KUKA KRL program: MyProgram_076().src

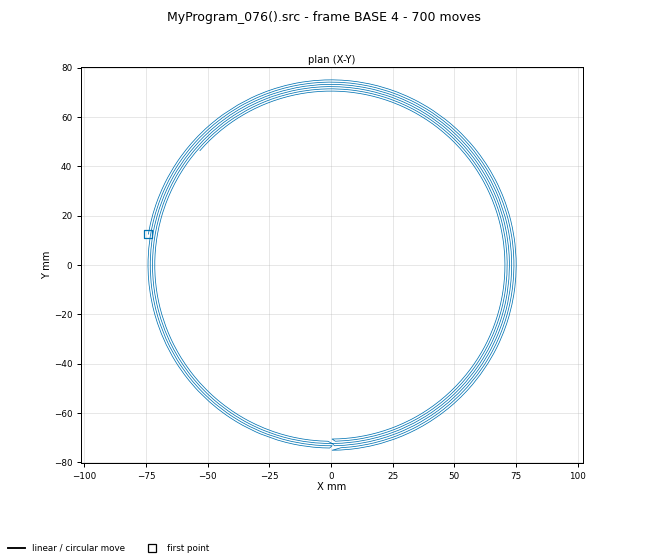
[picture p0: tool path of MyProgram_076().src in frame BASE 4, 700 of 700 moves have a stored position in this frame; points joined in program order, loops and branches not executed]
&ACCESS RVP
&REL 1
&PARAM TEMPLATE = C:\KRC\Roboter\Template\vorgabe
&PARAM EDITMASK = *
DEF MyProgram_076()
; ---- Setting reference (Base) ----
$BASE = BASE_DATA[4]

; --------------------------
; ---- Setting tool (TCP) ----
$TOOL = TOOL_DATA[3]
; --------------------------

$VEL.CP = VEL_APROX_PRINT
Startdeposition()
$VEL.CP = VEL_PRINT
LIN {X -74.0338,Y 12.5414,Z 79,A 163.3796,B 24.8998,C -2.3111,E1 24.8428,E2 281.1922} C_DIS
LIN {X -73.2521,Y 16.5095,Z 79,A 161.2903,B 24.8969,C -2.3435,E1 24.844,E2 283.2162} C_DIS
LIN {X -72.1494,Y 20.8052,Z 79,A 158.1049,B 24.8956,C -2.3587,E1 24.8463,E2 286.3839} C_DIS
LIN {X -70.9389,Y 24.6173,Z 79,A 155.0379,B 24.8948,C -2.3677,E1 24.8489,E2 289.4469} C_DIS
LIN {X -70.0447,Y 27.057,Z 79,A 152.3998,B 24.8956,C -2.3586,E1 24.8515,E2 292.1217} C_DIS
LIN {X -68.6085,Y 30.5169,Z 79,A 149.1898,B 24.8956,C -2.3591,E1 24.8551,E2 295.3482} C_DIS
LIN {X -67.2388,Y 33.425,Z 79,A 147.2866,B 24.8938,C -2.379,E1 24.8574,E2 297.2143} C_DIS
LIN {X -66.1724,Y 35.491,Z 79,A 145.1905,B 24.894,C -2.3766,E1 24.8602,E2 299.3271} C_DIS
LIN {X -63.8148,Y 39.5728,Z 79,A 141.9536,B 24.8923,C -2.3952,E1 24.8648,E2 302.5364} C_DIS
LIN {X -62.0519,Y 42.2834,Z 79,A 139.6485,B 24.8914,C -2.4058,E1 24.8683,E2 304.8278} C_DIS
LIN {X -60.8028,Y 44.0616,Z 79,A 137.7393,B 24.8915,C -2.4043,E1 24.8714,E2 306.7497} C_DIS
LIN {X -58.7303,Y 46.7866,Z 79,A 135.0507,B 24.8911,C -2.4094,E1 24.876,E2 309.4388} C_DIS
LIN {X -56.5657,Y 49.3821,Z 79,A 132.3745,B 24.8907,C -2.4137,E1 24.8809,E2 312.1171} C_DIS
LIN {X -53.9325,Y 52.2455,Z 79,A 129.4614,B 24.8899,C -2.4222,E1 24.8864,E2 315.0225} C_DIS
LIN {X -50.9748,Y 55.1346,Z 79,A 126.5258,B 24.8887,C -2.4348,E1 24.8923,E2 317.9402} C_DIS
LIN {X -49.0445,Y 56.8585,Z 79,A 124.2457,B 24.889,C -2.432,E1 24.8972,E2 320.2362} C_DIS
LIN {X -45.9844,Y 59.3611,Z 79,A 121.4566,B 24.8879,C -2.4439,E1 24.9032,E2 323.0073} C_DIS
LIN {X -43.6877,Y 61.071,Z 79,A 118.8455,B 24.8884,C -2.438,E1 24.9092,E2 325.6414} C_DIS
LIN {X -37.719,Y 64.9268,Z 79,A 113.8884,B 24.8865,C -2.4594,E1 24.9208,E2 330.5633} C_DIS
LIN {X -32.3398,Y 67.7676,Z 79,A 109.0548,B 24.8862,C -2.4622,E1 24.9328,E2 335.4033} C_DIS
LIN {X -30.0073,Y 68.8319,Z 79,A 106.5716,B 24.8871,C -2.4521,E1 24.9392,E2 337.9164} C_DIS
LIN {X -26.1038,Y 70.4061,Z 79,A 103.4974,B 24.8864,C -2.4597,E1 24.9472,E2 340.979} C_DIS
LIN {X -22.65,Y 71.5922,Z 79,A 100.0527,B 24.8877,C -2.4467,E1 24.9565,E2 344.461} C_DIS
LIN {X -18.3648,Y 72.8088,Z 79,A 96.6299,B 24.8874,C -2.4494,E1 24.9657,E2 347.8821} C_DIS
LIN {X -13.9688,Y 73.778,Z 79,A 94.2298,B 24.8847,C -2.4781,E1 24.9721,E2 350.2167} C_DIS
LIN {X -11.4549,Y 74.2095,Z 79,A 92.0843,B 24.8851,C -2.4744,E1 24.9781,E2 352.3729} C_DIS
LIN {X -6.9976,Y 74.7617,Z 79,A 87.808,B 24.8869,C -2.4547,E1 24.9901,E2 356.6986} C_DIS
LIN {X -2.4864,Y 75.0475,Z 79,A 85.4114,B 24.8843,C -2.4827,E1 24.9966,E2 359.0291} C_DIS
LIN {X 0.7273,Y 75.0854,Z 79,A 82.8148,B 24.8846,C -2.4794,E1 25.0039,E2 361.6334} C_DIS
LIN {X 4.3078,Y 74.9649,Z 79,A 79.597,B 24.8858,C -2.467,E1 25.0129,E2 364.8796} C_DIS
LIN {X 7.625,Y 74.7005,Z 79,A 77.7484,B 24.8841,C -2.4847,E1 25.0179,E2 366.6849} C_DIS
LIN {X 11.0283,Y 74.2755,Z 79,A 74.5426,B 24.8856,C -2.4686,E1 25.0269,E2 369.9263} C_DIS
LIN {X 15.5826,Y 73.4542,Z 79,A 71.3552,B 24.8849,C -2.4762,E1 25.0356,E2 373.0918} C_DIS
LIN {X 19.0638,Y 72.6291,Z 79,A 68.6928,B 24.8849,C -2.4764,E1 25.0428,E2 375.7498} C_DIS
LIN {X 23.5565,Y 71.2992,Z 79,A 65.0604,B 24.8853,C -2.4722,E1 25.0525,E2 379.3857} C_DIS
LIN {X 26.7438,Y 70.1646,Z 79,A 61.6181,B 24.8877,C -2.4466,E1 25.0616,E2 382.8812} C_DIS
LIN {X 30.9008,Y 68.4355,Z 79,A 59.2126,B 24.8854,C -2.4707,E1 25.0676,E2 385.2236} C_DIS
LIN {X 33.9507,Y 66.9752,Z 79,A 56.6895,B 24.8856,C -2.4691,E1 25.0739,E2 387.7438} C_DIS
LIN {X 35.7546,Y 66.0294,Z 79,A 54.9592,B 24.8862,C -2.4622,E1 25.0782,E2 389.4855} C_DIS
LIN {X 39.1193,Y 64.0934,Z 79,A 52.1395,B 24.8862,C -2.4619,E1 25.0849,E2 392.2974} C_DIS
LIN {X 41.3094,Y 62.7041,Z 79,A 49.8554,B 24.8873,C -2.4503,E1 25.0903,E2 394.6014} C_DIS
LIN {X 46.3215,Y 59.0989,Z 79,A 45.5003,B 24.8872,C -2.4521,E1 25.1001,E2 398.9366} C_DIS
LIN {X 48.4243,Y 57.3889,Z 79,A 42.7997,B 24.8891,C -2.4304,E1 25.1059,E2 401.6781} C_DIS
LIN {X 50.9296,Y 55.1769,Z 79,A 40.8978,B 24.8879,C -2.4436,E1 25.1098,E2 403.5411} C_DIS
LIN {X 52.8577,Y 53.3324,Z 79,A 38.5166,B 24.8892,C -2.4296,E1 25.1145,E2 405.9455} C_DIS
LIN {X 56.4292,Y 49.5384,Z 79,A 34.9262,B 24.889,C -2.4318,E1 25.1213,E2 409.5149} C_DIS
LIN {X 58.3316,Y 47.2832,Z 79,A 32.0216,B 24.8912,C -2.4079,E1 25.1265,E2 412.4626} C_DIS
LIN {X 60.4304,Y 44.5702,Z 79,A 29.7878,B 24.8908,C -2.4125,E1 25.1302,E2 414.6748} C_DIS
LIN {X 62.9223,Y 40.9777,Z 79,A 26.7139,B 24.8908,C -2.4116,E1 25.1349,E2 417.7354} C_DIS
LIN {X 64.6181,Y 38.2462,Z 79,A 23.7768,B 24.8927,C -2.3912,E1 25.1392,E2 420.7057} C_DIS
LIN {X 66.7813,Y 34.3302,Z 79,A 20.9154,B 24.8921,C -2.398,E1 25.1429,E2 423.536} C_DIS
LIN {X 67.7546,Y 32.3668,Z 79,A 19.0536,B 24.893,C -2.3878,E1 25.1452,E2 425.4119} C_DIS
LIN {X 69.485,Y 28.4629,Z 79,A 15.3261,B 24.8951,C -2.3649,E1 25.1493,E2 429.1731} C_DIS
LIN {X 70.7518,Y 25.1506,Z 79,A 13.3493,B 24.8939,C -2.3783,E1 25.1511,E2 431.1071} C_DIS
LIN {X 72.1899,Y 20.6623,Z 79,A 9.7524,B 24.8948,C -2.3676,E1 25.1541,E2 434.7089} C_DIS
LIN {X 72.8382,Y 18.2504,Z 79,A 7.2574,B 24.8969,C -2.3445,E1 25.1558,E2 437.2441} C_DIS
LIN {X 73.5531,Y 15.1069,Z 79,A 4.9587,B 24.8971,C -2.3417,E1 25.1571,E2 439.536} C_DIS
LIN {X 74.3323,Y 10.6297,Z 79,A 1.971,B 24.8968,C -2.3451,E1 25.1584,E2 442.4982} C_DIS
LIN {X 74.5961,Y 8.5861,Z 79,A 0.0072,B 24.8983,C -2.3286,E1 25.159,E2 444.4893} C_DIS
LIN {X 75.0392,Y 2.7571,Z 79,A -4.02,B 24.8983,C -2.3273,E1 25.1597,E2 448.4957} C_DIS
LIN {X 75.0885,Y -0.2198,Z 79,A -6.074,B 24.8984,C -2.3266,E1 25.1597,E2 450.5391} C_DIS
LIN {X 74.9286,Y -4.8989,Z 79,A -10.2294,B 24.9009,C -2.2979,E1 25.1592,E2 454.7376} C_DIS
LIN {X 74.5301,Y -9.1497,Z 79,A -13.0627,B 24.9007,C -2.3001,E1 25.1584,E2 457.549} C_DIS
LIN {X 74.0928,Y -12.1884,Z 79,A -15.2797,B 24.9011,C -2.2964,E1 25.1575,E2 459.7616} C_DIS
LIN {X 73.3464,Y -16.0806,Z 79,A -18.5241,B 24.9024,C -2.2803,E1 25.1556,E2 463.0251} C_DIS
LIN {X 72.2095,Y -20.593,Z 79,A -21.5023,B 24.9019,C -2.2862,E1 25.1536,E2 465.9721} C_DIS
LIN {X 71.233,Y -23.7528,Z 79,A -24.7017,B 24.9043,C -2.2583,E1 25.1508,E2 469.2193} C_DIS
LIN {X 69.9926,Y -27.1916,Z 79,A -27.419,B 24.9049,C -2.2519,E1 25.1481,E2 471.9366} C_DIS
LIN {X 68.3546,Y -31.0804,Z 79,A -30.3314,B 24.9049,C -2.2513,E1 25.1449,E2 474.8343} C_DIS
LIN {X 67.0986,Y -33.7059,Z 79,A -32.5046,B 24.9054,C -2.2462,E1 25.1422,E2 477.0081} C_DIS
LIN {X 65.901,Y -35.9913,Z 79,A -34.7495,B 24.9065,C -2.2323,E1 25.1392,E2 479.274} C_DIS
LIN {X 63.5951,Y -39.9245,Z 79,A -37.8445,B 24.9064,C -2.2337,E1 25.1348,E2 482.3497} C_DIS
LIN {X 60.5065,Y -44.4663,Z 79,A -42.0028,B 24.9073,C -2.2232,E1 25.1282,E2 486.5126} C_DIS
LIN {X 57.3809,Y -48.4337,Z 79,A -46.0102,B 24.9085,C -2.2086,E1 25.1212,E2 490.5358} C_DIS
LIN {X 55.3733,Y -50.7157,Z 79,A -48.5588,B 24.9095,C -2.1961,E1 25.1164,E2 493.1027} C_DIS
LIN {X 52.6657,Y -53.5221,Z 79,A -51.2668,B 24.9095,C -2.1966,E1 25.1111,E2 495.7979} C_DIS
LIN {X 49.7882,Y -56.21,Z 79,A -54.281,B 24.9101,C -2.1894,E1 25.1049,E2 498.817} C_DIS
LIN {X 47.4391,Y -58.2052,Z 79,A -56.8567,B 24.911,C -2.1778,E1 25.0993,E2 501.4103} C_DIS
LIN {X 44.4713,Y -60.5028,Z 79,A -59.6425,B 24.9113,C -2.174,E1 25.0931,E2 504.1949} C_DIS
LIN {X 40.3486,Y -63.3271,Z 79,A -63.2381,B 24.9114,C -2.1728,E1 25.0847,E2 507.7815} C_DIS
LIN {X 37.2123,Y -65.2193,Z 79,A -66.1227,B 24.9121,C -2.1652,E1 25.0778,E2 510.6753} C_DIS
LIN {X 34.3967,Y -66.7473,Z 79,A -68.4125,B 24.9121,C -2.1654,E1 25.0721,E2 512.9579} C_DIS
LIN {X 31.8505,Y -67.9989,Z 79,A -70.53,B 24.9122,C -2.1633,E1 25.0668,E2 515.0748} C_DIS
LIN {X 28.6942,Y -69.3901,Z 79,A -73.5255,B 24.9134,C -2.1493,E1 25.0591,E2 518.0965} C_DIS
LIN {X 25.511,Y -70.6223,Z 79,A -76.2197,B 24.9138,C -2.1434,E1 25.052,E2 520.7991} C_DIS
LIN {X 20.0691,Y -72.358,Z 79,A -80.4465,B 24.9139,C -2.1421,E1 25.0407,E2 525.0216} C_DIS
LIN {X 15.8281,Y -73.4015,Z 79,A -83.441,B 24.9134,C -2.1482,E1 25.0326,E2 527.9972} C_DIS
LIN {X 11.2138,Y -74.2468,Z 79,A -87.0755,B 24.9138,C -2.144,E1 25.0226,E2 531.638} C_DIS
LIN {X 8.1036,Y -74.6504,Z 79,A -89.4305,B 24.9138,C -2.1435,E1 25.0161,E2 533.9922} C_DIS
LIN {X 3.8663,Y -74.9893,Z 79,A -93.5069,B 24.9157,C -2.1198,E1 25.0045,E2 538.1233} C_DIS
LIN {X 0.4928,Y -75.0785,Z 79,A -93.6611,B 24.9105,C -2.1847,E1 25.0046,E2 538.1233} C_DIS
Enddeposition()
LIN {X 0.4928,Y -75.0785,Z 79,A -93.6611,B 24.9105,C -2.1847,E1 25.0046,E2 538.1233} C_DIS
Startdeposition()
$VEL.CP = VEL_PRINT
LIN {X 4.0815,Y -74.0642,Z 79,A -91.2785,B 24.91,C -2.1904,E1 25.0112,E2 535.7279} C_DIS
LIN {X 8.0955,Y -73.7344,Z 79,A -88.3098,B 24.9102,C -2.1882,E1 25.0195,E2 532.7665} C_DIS
LIN {X 11.0368,Y -73.3515,Z 79,A -85.1411,B 24.908,C -2.2141,E1 25.0284,E2 529.5392} C_DIS
LIN {X 14.9582,Y -72.6527,Z 79,A -83.3262,B 24.9107,C -2.1816,E1 25.0331,E2 527.8034} C_DIS
LIN {X 17.5684,Y -72.066,Z 79,A -80.6303,B 24.9091,C -2.201,E1 25.0406,E2 525.0653} C_DIS
LIN {X 21.3791,Y -71.0295,Z 79,A -77.0856,B 24.9077,C -2.2184,E1 25.0502,E2 521.4856} C_DIS
LIN {X 24.874,Y -69.8824,Z 79,A -75.2446,B 24.9097,C -2.1937,E1 25.0549,E2 519.7068} C_DIS
LIN {X 26.7368,Y -69.1907,Z 79,A -73.4018,B 24.9088,C -2.2044,E1 25.0597,E2 517.8425} C_DIS
LIN {X 30.013,Y -67.8347,Z 79,A -70.6724,B 24.9085,C -2.2081,E1 25.0667,E2 515.1108} C_DIS
LIN {X 33.3671,Y -66.2483,Z 79,A -68.1884,B 24.9091,C -2.2019,E1 25.0729,E2 512.6482} C_DIS
LIN {X 34.9862,Y -65.4087,Z 79,A -66.3095,B 24.9077,C -2.2177,E1 25.0776,E2 510.7373} C_DIS
LIN {X 38.5939,Y -63.3457,Z 79,A -63.4619,B 24.9081,C -2.2131,E1 25.0844,E2 507.9092} C_DIS
LIN {X 40.1525,Y -62.3694,Z 79,A -61.5131,B 24.9066,C -2.231,E1 25.0891,E2 505.9243} C_DIS
LIN {X 43.2174,Y -60.2863,Z 79,A -59.2432,B 24.9076,C -2.2196,E1 25.0942,E2 503.6892} C_DIS
LIN {X 45.6157,Y -58.4925,Z 79,A -56.4487,B 24.906,C -2.2385,E1 25.1005,E2 500.8603} C_DIS
LIN {X 48.7088,Y -55.943,Z 79,A -53.2307,B 24.9051,C -2.2489,E1 25.1073,E2 497.63} C_DIS
LIN {X 52.1516,Y -52.7482,Z 79,A -49.8965,B 24.9051,C -2.2489,E1 25.114,E2 494.3098} C_DIS
LIN {X 55.2474,Y -49.4963,Z 79,A -46.6042,B 24.9048,C -2.2523,E1 25.1203,E2 491.0238} C_DIS
LIN {X 59.3132,Y -44.5433,Z 79,A -41.5957,B 24.9036,C -2.267,E1 25.1291,E2 486.004} C_DIS
LIN {X 61.9752,Y -40.7583,Z 79,A -38.3749,B 24.9036,C -2.2663,E1 25.1341,E2 482.8006} C_DIS
LIN {X 63.2688,Y -38.7198,Z 79,A -35.4397,B 24.9004,C -2.3035,E1 25.1385,E2 479.7924} C_DIS
LIN {X 65.1878,Y -35.3937,Z 79,A -33.2931,B 24.9018,C -2.2875,E1 25.1414,E2 477.6947} C_DIS
LIN {X 66.848,Y -32.1483,Z 79,A -30.413,B 24.9009,C -2.2977,E1 25.1449,E2 474.806} C_DIS
LIN {X 68.2757,Y -28.9936,Z 79,A -27.8103,B 24.9004,C -2.3036,E1 25.1478,E2 472.2036} C_DIS
LIN {X 69.318,Y -26.4046,Z 79,A -25.8859,B 24.9004,C -2.3033,E1 25.1498,E2 470.2906} C_DIS
LIN {X 70.6962,Y -22.4547,Z 79,A -22.6503,B 24.8996,C -2.3133,E1 25.1527,E2 467.0496} C_DIS
LIN {X 71.4938,Y -19.7737,Z 79,A -20.1823,B 24.8982,C -2.3293,E1 25.1546,E2 464.558} C_DIS
LIN {X 72.4055,Y -16.1152,Z 79,A -16.8313,B 24.8962,C -2.3517,E1 25.1567,E2 461.1737} C_DIS
LIN {X 73.0556,Y -12.8498,Z 79,A -15.2572,B 24.8982,C -2.3298,E1 25.1575,E2 459.6603} C_DIS
LIN {X 73.5866,Y -9.3387,Z 79,A -11.8884,B 24.8957,C -2.3573,E1 25.1588,E2 456.2465} C_DIS
LIN {X 74.0023,Y -5.0821,Z 79,A -7.8424,B 24.8928,C -2.3903,E1 25.1597,E2 452.1466} C_DIS
LIN {X 74.1745,Y -0.5549,Z 79,A -5.6994,B 24.8954,C -2.3605,E1 25.1597,E2 450.0866} C_DIS
LIN {X 74.1537,Y 1.884,Z 79,A -2.7613,B 24.8921,C -2.3982,E1 25.1596,E2 447.0771} C_DIS
LIN {X 73.9615,Y 5.6506,Z 79,A -0.6692,B 24.8935,C -2.3826,E1 25.1592,E2 445.034} C_DIS
LIN {X 73.6238,Y 9.0483,Z 79,A 1.7052,B 24.8935,C -2.383,E1 25.1585,E2 442.6727} C_DIS
LIN {X 73.2988,Y 11.3776,Z 79,A 3.9459,B 24.8918,C -2.4014,E1 25.1575,E2 440.4019} C_DIS
LIN {X 72.654,Y 14.9521,Z 79,A 6.6534,B 24.8913,C -2.4071,E1 25.1561,E2 437.6968} C_DIS
LIN {X 71.7299,Y 18.8993,Z 79,A 9.4116,B 24.8914,C -2.4055,E1 25.1543,E2 434.9583} C_DIS
LIN {X 70.995,Y 21.4902,Z 79,A 12.4708,B 24.8882,C -2.4409,E1 25.1518,E2 431.8329} C_DIS
LIN {X 69.8305,Y 25.0208,Z 79,A 15.0646,B 24.8882,C -2.4409,E1 25.1493,E2 429.2536} C_DIS
LIN {X 68.3042,Y 28.926,Z 79,A 17.6554,B 24.8891,C -2.431,E1 25.1467,E2 426.7004} C_DIS
LIN {X 66.6033,Y 32.6537,Z 79,A 20.616,B 24.8888,C -2.4339,E1 25.1432,E2 423.7491} C_DIS
LIN {X 65.4425,Y 34.9229,Z 79,A 23.6796,B 24.8854,C -2.4714,E1 25.1391,E2 420.6128} C_DIS
LIN {X 63.5934,Y 38.1864,Z 79,A 25.5376,B 24.8875,C -2.4485,E1 25.1365,E2 418.8186} C_DIS
LIN {X 61.4007,Y 41.6186,Z 79,A 28.8611,B 24.8863,C -2.4617,E1 25.1315,E2 415.4806} C_DIS
LIN {X 57.9026,Y 46.3622,Z 79,A 33.2981,B 24.8856,C -2.4693,E1 25.124,E2 411.0468} C_DIS
LIN {X 56.602,Y 47.9418,Z 79,A 35.7497,B 24.8829,C -2.4982,E1 25.1195,E2 408.538} C_DIS
LIN {X 54.2039,Y 50.6363,Z 79,A 38.0338,B 24.8837,C -2.4897,E1 25.1152,E2 406.2839} C_DIS
LIN {X 51.9222,Y 52.9748,Z 79,A 40.2849,B 24.8839,C -2.4872,E1 25.1108,E2 404.0484} C_DIS
LIN {X 48.6804,Y 55.9679,Z 79,A 44.1161,B 24.8821,C -2.506,E1 25.1027,E2 400.188} C_DIS
LIN {X 45.196,Y 58.8174,Z 79,A 47.4692,B 24.8819,C -2.5087,E1 25.0954,E2 396.8409} C_DIS
LIN {X 41.1343,Y 61.7273,Z 79,A 50.8713,B 24.8825,C -2.5022,E1 25.0877,E2 393.4659} C_DIS
LIN {X 38.8606,Y 63.1836,Z 79,A 53.3129,B 24.8812,C -2.5153,E1 25.0818,E2 391.001} C_DIS
LIN {X 34.5422,Y 65.643,Z 79,A 56.6631,B 24.882,C -2.507,E1 25.0737,E2 387.6805} C_DIS
LIN {X 32.2302,Y 66.8086,Z 79,A 58.7379,B 24.8816,C -2.5115,E1 25.0685,E2 385.6004} C_DIS
LIN {X 27.2296,Y 68.998,Z 79,A 62.9805,B 24.8811,C -2.5166,E1 25.0576,E2 381.3556} C_DIS
LIN {X 23.4337,Y 70.3783,Z 79,A 65.8887,B 24.8814,C -2.5136,E1 25.05,E2 378.4606} C_DIS
LIN {X 18.3849,Y 71.8621,Z 79,A 69.6829,B 24.8818,C -2.5091,E1 25.0399,E2 374.6836} C_DIS
LIN {X 15.2731,Y 72.5867,Z 79,A 72.8346,B 24.88,C -2.5287,E1 25.0312,E2 371.4897} C_DIS
LIN {X 11.7393,Y 73.2412,Z 79,A 75.7304,B 24.8796,C -2.5328,E1 25.0232,E2 368.5871} C_DIS
LIN {X 7.9492,Y 73.7497,Z 79,A 79.408,B 24.8777,C -2.5527,E1 25.0129,E2 364.8648} C_DIS
LIN {X 3.7851,Y 74.0806,Z 79,A 81.4299,B 24.8807,C -2.5207,E1 25.0075,E2 362.9199} C_DIS
LIN {X -0.7943,Y 74.1731,Z 79,A 84.9826,B 24.8807,C -2.5205,E1 24.9976,E2 359.368} C_DIS
LIN {X -4.5442,Y 74.0386,Z 79,A 88.5493,B 24.8792,C -2.5369,E1 24.9875,E2 355.7614} C_DIS
LIN {X -8.3481,Y 73.7058,Z 79,A 91.3267,B 24.8798,C -2.5309,E1 24.9798,E2 352.9967} C_DIS
LIN {X -12.706,Y 73.0815,Z 79,A 94.2335,B 24.8812,C -2.5159,E1 24.9719,E2 350.1231} C_DIS
LIN {X -15.6953,Y 72.4971,Z 79,A 97.1755,B 24.8799,C -2.529,E1 24.9637,E2 347.1464} C_DIS
LIN {X -18.9763,Y 71.7089,Z 79,A 100.1883,B 24.8792,C -2.5368,E1 24.9555,E2 344.1107} C_DIS
LIN {X -22.4216,Y 70.708,Z 79,A 101.9844,B 24.8818,C -2.509,E1 24.9509,E2 342.3777} C_DIS
LIN {X -26.7617,Y 69.1818,Z 79,A 105.6431,B 24.882,C -2.5071,E1 24.9413,E2 338.716} C_DIS
LIN {X -30.2247,Y 67.74,Z 79,A 108.6639,B 24.8821,C -2.506,E1 24.9335,E2 335.6908} C_DIS
LIN {X -35.1702,Y 65.309,Z 79,A 112.9042,B 24.8828,C -2.4988,E1 24.923,E2 331.4564} C_DIS
LIN {X -36.9477,Y 64.3197,Z 79,A 115.711,B 24.8802,C -2.5266,E1 24.916,E2 328.5749} C_DIS
LIN {X -40.9698,Y 61.8358,Z 79,A 117.5481,B 24.885,C -2.4752,E1 24.912,E2 326.8545} C_DIS
LIN {X -43.9498,Y 59.7545,Z 79,A 121.126,B 24.8838,C -2.4882,E1 24.9037,E2 323.2333} C_DIS
LIN {X -47.2986,Y 57.1402,Z 79,A 124.7937,B 24.8836,C -2.4905,E1 24.8957,E2 319.5463} C_DIS
LIN {X -49.7901,Y 54.9844,Z 79,A 127.0934,B 24.8847,C -2.4788,E1 24.891,E2 317.2653} C_DIS
LIN {X -53.273,Y 51.6157,Z 79,A 130.5791,B 24.8861,C -2.4638,E1 24.8841,E2 313.8009} C_DIS
LIN {X -55.111,Y 49.6487,Z 79,A 133.1468,B 24.8855,C -2.4703,E1 24.8792,E2 311.2063} C_DIS
LIN {X -57.2689,Y 47.144,Z 79,A 135.819,B 24.8858,C -2.4665,E1 24.8744,E2 308.5307} C_DIS
LIN {X -60.1199,Y 43.4507,Z 79,A 138.8407,B 24.888,C -2.4431,E1 24.8694,E2 305.5504} C_DIS
LIN {X -62.0554,Y 40.6361,Z 79,A 141.7341,B 24.888,C -2.4419,E1 24.8649,E2 302.6454} C_DIS
LIN {X -64.0387,Y 37.4342,Z 79,A 144.6852,B 24.8888,C -2.4347,E1 24.8607,E2 299.6965} C_DIS
LIN {X -65.7699,Y 34.3013,Z 79,A 147.5541,B 24.8893,C -2.4291,E1 24.8569,E2 296.8256} C_DIS
LIN {X -67.7277,Y 30.252,Z 79,A 150.5611,B 24.8912,C -2.4079,E1 24.8534,E2 293.8528} C_DIS
LIN {X -68.4138,Y 28.666,Z 79,A 152.9679,B 24.8893,C -2.429,E1 24.8507,E2 291.3822} C_DIS
LIN {X -69.7897,Y 25.1327,Z 79,A 155.0915,B 24.8918,C -2.4012,E1 24.8487,E2 289.3132} C_DIS
LIN {X -71.1483,Y 20.9785,Z 79,A 158.2409,B 24.8932,C -2.3855,E1 24.8461,E2 286.1831} C_DIS
LIN {X -72.0044,Y 17.8206,Z 79,A 161.0875,B 24.8932,C -2.385,E1 24.8441,E2 283.3212} C_DIS
LIN {X -72.8749,Y 13.8365,Z 79,A 163.9856,B 24.8947,C -2.3692,E1 24.8424,E2 280.4436} C_DIS
LIN {X -73.2957,Y 11.3974,Z 79,A 167.3016,B 24.8923,C -2.3961,E1 24.841,E2 277.0438} C_DIS
LIN {X -73.871,Y 6.7269,Z 79,A 169.1745,B 24.897,C -2.3434,E1 24.8405,E2 275.2855} C_DIS
LIN {X -74.1464,Y 2.1214,Z 79,A 173.2157,B 24.897,C -2.343,E1 24.8398,E2 271.2209} C_DIS
LIN {X -74.1742,Y -0.6115,Z 79,A 175.7277,B 24.8968,C -2.3456,E1 24.8398,E2 268.6876} C_DIS
LIN {X -74.0549,Y -4.2498,Z 79,A 179.1346,B 24.8963,C -2.3507,E1 24.8403,E2 265.248} C_DIS
LIN {X -73.7532,Y -7.9161,Z 79,A -179.282,B 24.8997,C -2.3124,E1 24.8407,E2 263.7467} C_DIS
LIN {X -73.1849,Y -12.0896,Z 79,A -175.4813,B 24.8995,C -2.3149,E1 24.8422,E2 259.9172} C_DIS
LIN {X -72.2272,Y -16.8949,Z 79,A -172.3249,B 24.9017,C -2.2887,E1 24.844,E2 256.8049} C_DIS
LIN {X -71.3757,Y -20.1903,Z 79,A -168.36,B 24.8997,C -2.3121,E1 24.8469,E2 252.761} C_DIS
LIN {X -70.3615,Y -23.4834,Z 79,A -166.3916,B 24.9018,C -2.2878,E1 24.8486,E2 250.8392} C_DIS
LIN {X -68.727,Y -27.9063,Z 79,A -162.4807,B 24.9022,C -2.2837,E1 24.8525,E2 246.9163} C_DIS
LIN {X -66.7431,Y -32.3666,Z 79,A -158.4217,B 24.9025,C -2.28,E1 24.8573,E2 242.8439} C_DIS
LIN {X -64.3289,Y -36.9318,Z 79,A -155.0585,B 24.9047,C -2.2544,E1 24.8618,E2 239.5242} C_DIS
LIN {X -63.0078,Y -39.1435,Z 79,A -153.3025,B 24.9056,C -2.2436,E1 24.8643,E2 237.7849} C_DIS
LIN {X -61.7944,Y -41.0326,Z 79,A -150.1498,B 24.903,C -2.2735,E1 24.8693,E2 234.5451} C_DIS
LIN {X -59.3355,Y -44.5136,Z 79,A -147.9554,B 24.906,C -2.2388,E1 24.8728,E2 232.4229} C_DIS
LIN {X -57.5612,Y -46.7855,Z 79,A -144.7691,B 24.9044,C -2.257,E1 24.8785,E2 229.1782} C_DIS
LIN {X -55.0659,Y -49.6991,Z 79,A -142.8721,B 24.9072,C -2.2243,E1 24.8819,E2 227.3508} C_DIS
LIN {X -53.786,Y -51.0819,Z 79,A -140.6203,B 24.9058,C -2.2406,E1 24.8863,E2 225.0501} C_DIS
LIN {X -49.2763,Y -55.4444,Z 79,A -136.2549,B 24.9076,C -2.219,E1 24.8951,E2 220.7186} C_DIS
LIN {X -45.8359,Y -58.3204,Z 79,A -132.4378,B 24.9074,C -2.2214,E1 24.9035,E2 216.8812} C_DIS
LIN {X -42.8027,Y -60.5823,Z 79,A -130.1365,B 24.9091,C -2.201,E1 24.9086,E2 214.6206} C_DIS
LIN {X -41.0359,Y -61.7922,Z 79,A -127.9596,B 24.9083,C -2.2115,E1 24.9137,E2 212.4115} C_DIS
LIN {X -38.4374,Y -63.4408,Z 79,A -125.8461,B 24.9091,C -2.2013,E1 24.9187,E2 210.3156} C_DIS
LIN {X -35.8228,Y -64.9541,Z 79,A -123.4379,B 24.9092,C -2.2,E1 24.9245,E2 207.9034} C_DIS
LIN {X -30.5377,Y -67.5988,Z 79,A -119.1115,B 24.9102,C -2.1885,E1 24.9354,E2 203.5933} C_DIS
LIN {X -28.5665,Y -68.4557,Z 79,A -116.7849,B 24.9089,C -2.2039,E1 24.9414,E2 201.2245} C_DIS
LIN {X -21.7815,Y -70.9067,Z 79,A -111.876,B 24.9107,C -2.1821,E1 24.9543,E2 196.3582} C_DIS
LIN {X -18.2713,Y -71.8903,Z 79,A -108.7906,B 24.9103,C -2.1874,E1 24.9626,E2 193.2554} C_DIS
LIN {X -15.1008,Y -72.6229,Z 79,A -106.2106,B 24.9103,C -2.188,E1 24.9697,E2 190.6708} C_DIS
LIN {X -12.3519,Y -73.141,Z 79,A -104.1832,B 24.9106,C -2.1837,E1 24.9752,E2 188.6514} C_DIS
LIN {X -7.0887,Y -73.8376,Z 79,A -100.1371,B 24.9107,C -2.1816,E1 24.9865,E2 184.6076} C_DIS
LIN {X -3.4251,Y -74.0978,Z 79,A -97.3242,B 24.9107,C -2.181,E1 24.9943,E2 181.7952} C_DIS
LIN {X -0.5354,Y -74.1747,Z 79,A -93.8754,B 24.908,C -2.2146,E1 25.0042,E2 178.2666} C_DIS
LIN {X -0.5354,Y -74.1747,Z 79,A -93.8754,B 24.908,C -2.2146,E1 25.0042,E2 178.2666} C_DIS
Enddeposition()
LIN {X 0.469,Y -73.2518,Z 79,A -95.0565,B 24.911,C -2.1779,E1 25.0006,E2 179.5349} C_DIS
Startdeposition()
$VEL.CP = VEL_PRINT
LIN {X -2.1885,Y -73.232,Z 79,A -98.3137,B 24.9136,C -2.1468,E1 24.9913,E2 182.8662} C_DIS
LIN {X -6.0742,Y -73.0128,Z 79,A -100.1727,B 24.9111,C -2.1773,E1 24.9863,E2 184.6535} C_DIS
LIN {X -11.0273,Y -72.4303,Z 79,A -104.2061,B 24.9113,C -2.1745,E1 24.9751,E2 188.6964} C_DIS
LIN {X -16.045,Y -71.4875,Z 79,A -108.4932,B 24.9118,C -2.1685,E1 24.9633,E2 193.0025} C_DIS
LIN {X -19.7606,Y -70.5499,Z 79,A -111.3689,B 24.9114,C -2.1733,E1 24.9556,E2 195.871} C_DIS
LIN {X -25.5892,Y -68.6517,Z 79,A -116.4591,B 24.9117,C -2.1698,E1 24.9421,E2 200.9793} C_DIS
LIN {X -28.4071,Y -67.5333,Z 79,A -118.6089,B 24.9111,C -2.1776,E1 24.9366,E2 203.1152} C_DIS
LIN {X -33.0023,Y -65.4099,Z 79,A -122.7459,B 24.9111,C -2.1779,E1 24.9261,E2 207.2622} C_DIS
LIN {X -36.2952,Y -63.643,Z 79,A -125.765,B 24.9109,C -2.1794,E1 24.9187,E2 210.2864} C_DIS
LIN {X -39.9067,Y -61.4436,Z 79,A -128.8723,B 24.9101,C -2.1892,E1 24.9114,E2 213.3802} C_DIS
LIN {X -42.2551,Y -59.8528,Z 79,A -131.0563,B 24.9097,C -2.1936,E1 24.9064,E2 215.561} C_DIS
LIN {X -46.7553,Y -56.4062,Z 79,A -135.4753,B 24.9091,C -2.2019,E1 24.8967,E2 219.9767} C_DIS
LIN {X -49.2081,Y -54.2814,Z 79,A -137.7798,B 24.9082,C -2.2123,E1 24.8919,E2 222.2653} C_DIS
LIN {X -51.4486,Y -52.1609,Z 79,A -140.7512,B 24.9089,C -2.2041,E1 24.8859,E2 225.2689} C_DIS
LIN {X -53.738,Y -49.8003,Z 79,A -143.3532,B 24.9085,C -2.2089,E1 24.8809,E2 227.8707} C_DIS
LIN {X -56.0934,Y -47.1317,Z 79,A -145.8614,B 24.9074,C -2.2216,E1 24.8764,E2 230.36} C_DIS
LIN {X -58.0378,Y -44.7138,Z 79,A -148.396,B 24.9071,C -2.2248,E1 24.872,E2 232.8988} C_DIS
LIN {X -60.8443,Y -40.8141,Z 79,A -152.0295,B 24.9061,C -2.237,E1 24.8662,E2 236.5212} C_DIS
LIN {X -62.3525,Y -38.4713,Z 79,A -154.3932,B 24.9061,C -2.2383,E1 24.8627,E2 238.8937} C_DIS
LIN {X -65.3459,Y -33.1313,Z 79,A -159.08,B 24.9047,C -2.2535,E1 24.8564,E2 243.569} C_DIS
LIN {X -66.9238,Y -29.8148,Z 79,A -162.2056,B 24.9045,C -2.2558,E1 24.8527,E2 246.7063} C_DIS
LIN {X -69.1561,Y -24.1898,Z 79,A -166.4897,B 24.9025,C -2.2796,E1 24.8485,E2 250.9576} C_DIS
LIN {X -70.1732,Y -21.0593,Z 79,A -169.3838,B 24.9025,C -2.28,E1 24.846,E2 253.8674} C_DIS
LIN {X -71.0715,Y -17.7977,Z 79,A -172.0317,B 24.9018,C -2.2879,E1 24.8442,E2 256.5119} C_DIS
LIN {X -71.9666,Y -13.7309,Z 79,A -175.7505,B 24.9018,C -2.2876,E1 24.8421,E2 260.2533} C_DIS
LIN {X -72.6762,Y -9.2688,Z 79,A -178.8083,B 24.9,C -2.3092,E1 24.8409,E2 263.2778} C_DIS
LIN {X -72.9268,Y -7.0342,Z 79,A 178.9602,B 24.9004,C -2.3041,E1 24.8403,E2 265.5347} C_DIS
LIN {X -73.2448,Y -1.7539,Z 79,A 175.2001,B 24.8985,C -2.3256,E1 24.8398,E2 269.2662} C_DIS
LIN {X -73.2496,Y 1.4929,Z 79,A 172.6783,B 24.8978,C -2.334,E1 24.8398,E2 271.783} C_DIS
LIN {X -72.9863,Y 6.3903,Z 79,A 169.1514,B 24.8961,C -2.3531,E1 24.8405,E2 275.2855} C_DIS
LIN {X -72.5078,Y 10.5062,Z 79,A 165.6047,B 24.8958,C -2.3565,E1 24.8417,E2 278.8452} C_DIS
LIN {X -72.0376,Y 13.3586,Z 79,A 163.2226,B 24.8954,C -2.361,E1 24.8428,E2 281.2309} C_DIS
LIN {X -71.5383,Y 15.8122,Z 79,A 161.0326,B 24.8954,C -2.362,E1 24.8441,E2 283.4314} C_DIS
LIN {X -70.4093,Y 20.2568,Z 79,A 158.0164,B 24.8932,C -2.3859,E1 24.8463,E2 286.408} C_DIS
LIN {X -69.5966,Y 22.8941,Z 79,A 155.2853,B 24.8937,C -2.3797,E1 24.8486,E2 289.1695} C_DIS
LIN {X -67.7277,Y 27.9428,Z 79,A 151.2702,B 24.8922,C -2.3969,E1 24.8526,E2 293.1662} C_DIS
LIN {X -66.6646,Y 30.3916,Z 79,A 149.0386,B 24.8919,C -2.3998,E1 24.8552,E2 295.403} C_DIS
LIN {X -65.0686,Y 33.6739,Z 79,A 146.3968,B 24.8907,C -2.413,E1 24.8584,E2 298.0275} C_DIS
LIN {X -63.8582,Y 35.9151,Z 79,A 144.334,B 24.8904,C -2.4171,E1 24.8612,E2 300.0913} C_DIS
LIN {X -62.4342,Y 38.3379,Z 79,A 141.781,B 24.8905,C -2.4153,E1 24.8649,E2 302.6619} C_DIS
LIN {X -59.3693,Y 42.9323,Z 79,A 136.744,B 24.8909,C -2.4109,E1 24.8731,E2 307.734} C_DIS
LIN {X -56.7859,Y 46.2939,Z 79,A 134.651,B 24.8876,C -2.4472,E1 24.8766,E2 309.7501} C_DIS
LIN {X -53.6253,Y 49.9209,Z 79,A 130.6608,B 24.8872,C -2.4514,E1 24.884,E2 313.7483} C_DIS
LIN {X -51.513,Y 52.0971,Z 79,A 127.8919,B 24.8875,C -2.448,E1 24.8895,E2 316.5372} C_DIS
LIN {X -48.7634,Y 54.6796,Z 79,A 124.2725,B 24.8883,C -2.4394,E1 24.8971,E2 320.1916} C_DIS
LIN {X -45.4892,Y 57.4322,Z 79,A 121.9155,B 24.8856,C -2.4693,E1 24.9021,E2 322.4861} C_DIS
LIN {X -40.7703,Y 60.8739,Z 79,A 117.6196,B 24.8841,C -2.4848,E1 24.9118,E2 326.7599} C_DIS
LIN {X -37.3264,Y 63.0433,Z 79,A 113.9811,B 24.8846,C -2.4799,E1 24.9204,E2 330.4215} C_DIS
LIN {X -34.0098,Y 64.8928,Z 79,A 111.0353,B 24.8841,C -2.4855,E1 24.9277,E2 333.3624} C_DIS
LIN {X -30.6416,Y 66.55,Z 79,A 108.292,B 24.8832,C -2.4946,E1 24.9345,E2 336.0909} C_DIS
LIN {X -26.618,Y 68.2585,Z 79,A 104.6302,B 24.8832,C -2.4935,E1 24.944,E2 339.7635} C_DIS
LIN {X -23.4771,Y 69.4013,Z 79,A 102.2704,B 24.8824,C -2.5029,E1 24.9502,E2 342.1057} C_DIS
LIN {X -19.5949,Y 70.5964,Z 79,A 98.9056,B 24.8825,C -2.5017,E1 24.9592,E2 345.4788} C_DIS
LIN {X -14.0869,Y 71.8981,Z 79,A 94.9342,B 24.8811,C -2.5169,E1 24.97,E2 349.4192} C_DIS
LIN {X -10.6551,Y 72.4866,Z 79,A 91.2208,B 24.8832,C -2.4943,E1 24.9803,E2 353.1898} C_DIS
LIN {X -4.9655,Y 73.0962,Z 79,A 86.8712,B 24.8827,C -2.4995,E1 24.9924,E2 357.529} C_DIS
LIN {X -1.3029,Y 73.2531,Z 79,A 83.3313,B 24.8842,C -2.4835,E1 25.0024,E2 361.1072} C_DIS
LIN {X 3.3116,Y 73.19,Z 79,A 81.0729,B 24.881,C -2.5178,E1 25.0085,E2 363.2836} C_DIS
LIN {X 8.2086,Y 72.8041,Z 79,A 76.6408,B 24.8825,C -2.5024,E1 25.0209,E2 367.7499} C_DIS
LIN {X 12.9447,Y 72.1121,Z 79,A 72.5939,B 24.8833,C -2.4934,E1 25.0321,E2 371.8139} C_DIS
LIN {X 16.2696,Y 71.4358,Z 79,A 70.634,B 24.8817,C -2.51,E1 25.0373,E2 373.7318} C_DIS
LIN {X 18.4099,Y 70.9142,Z 79,A 67.8706,B 24.8844,C -2.4819,E1 25.045,E2 376.5574} C_DIS
LIN {X 22.5638,Y 69.7036,Z 79,A 65.8034,B 24.8814,C -2.5138,E1 25.0503,E2 378.5454} C_DIS
LIN {X 25.3144,Y 68.7528,Z 79,A 63.2175,B 24.8824,C -2.5035,E1 25.0571,E2 381.1503} C_DIS
LIN {X 29.2001,Y 67.1942,Z 79,A 59.5793,B 24.8836,C -2.4905,E1 25.0665,E2 384.8109} C_DIS
LIN {X 33.0679,Y 65.3783,Z 79,A 56.5145,B 24.8833,C -2.4938,E1 25.0742,E2 387.8598} C_DIS
LIN {X 35.7581,Y 63.9459,Z 79,A 54.1625,B 24.8835,C -2.4914,E1 25.0799,E2 390.2106} C_DIS
LIN {X 38.5429,Y 62.3078,Z 79,A 51.7309,B 24.8835,C -2.4903,E1 25.0857,E2 392.6373} C_DIS
LIN {X 40.9585,Y 60.7465,Z 79,A 48.2218,B 24.8871,C -2.4527,E1 25.094,E2 396.2235} C_DIS
LIN {X 45.0766,Y 57.7582,Z 79,A 45.5503,B 24.8845,C -2.4811,E1 25.0998,E2 398.8182} C_DIS
LIN {X 48.1064,Y 55.2585,Z 79,A 42.1456,B 24.8859,C -2.4661,E1 25.1071,E2 402.2451} C_DIS
LIN {X 51.1574,Y 52.4483,Z 79,A 39.3728,B 24.8853,C -2.4725,E1 25.1127,E2 404.9913} C_DIS
LIN {X 52.7316,Y 50.8635,Z 79,A 36.4827,B 24.8885,C -2.4372,E1 25.1184,E2 407.9524} C_DIS
LIN {X 55.6738,Y 47.6253,Z 79,A 34.2216,B 24.8863,C -2.4617,E1 25.1224,E2 410.1456} C_DIS
LIN {X 58.0172,Y 44.7406,Z 79,A 30.9279,B 24.8879,C -2.4439,E1 25.1282,E2 413.4658} C_DIS
LIN {X 60.2532,Y 41.6809,Z 79,A 28.52,B 24.8871,C -2.4523,E1 25.132,E2 415.8422} C_DIS
LIN {X 62.4561,Y 38.3019,Z 79,A 25.0748,B 24.8886,C -2.4359,E1 25.1373,E2 419.3087} C_DIS
LIN {X 64.7684,Y 34.2459,Z 79,A 21.5807,B 24.8891,C -2.4307,E1 25.142,E2 422.7972} C_DIS
LIN {X 66.8935,Y 29.8837,Z 79,A 17.7143,B 24.8903,C -2.418,E1 25.1466,E2 426.6725} C_DIS
LIN {X 68.1096,Y 26.9972,Z 79,A 15.0241,B 24.8915,C -2.4042,E1 25.1495,E2 429.3807} C_DIS
LIN {X 70.623,Y 19.5007,Z 79,A 9.3481,B 24.8919,C -2.4005,E1 25.1543,E2 435.0333} C_DIS
LIN {X 71.3658,Y 16.5725,Z 79,A 6.7104,B 24.8932,C -2.3854,E1 25.1561,E2 437.6914} C_DIS
LIN {X 72.1151,Y 12.9277,Z 79,A 3.6181,B 24.8945,C -2.3711,E1 25.1577,E2 440.7992} C_DIS
LIN {X 72.6444,Y 9.5138,Z 79,A 0.929,B 24.8952,C -2.3631,E1 25.1587,E2 443.4915} C_DIS
LIN {X 73.0644,Y 5.4297,Z 79,A -2.1332,B 24.8957,C -2.3572,E1 25.1595,E2 446.5493} C_DIS
LIN {X 73.2612,Y 0.7918,Z 79,A -5.2472,B 24.8954,C -2.3607,E1 25.1598,E2 449.6366} C_DIS
LIN {X 73.2254,Y -2.4032,Z 79,A -8.5111,B 24.8981,C -2.3306,E1 25.1596,E2 452.9522} C_DIS
LIN {X 72.9966,Y -6.2774,Z 79,A -11.9795,B 24.9,C -2.3085,E1 25.1588,E2 456.4523} C_DIS
LIN {X 72.5395,Y -10.2827,Z 79,A -14.2357,B 24.8986,C -2.3243,E1 25.158,E2 458.6578} C_DIS
LIN {X 71.6792,Y -15.1644,Z 79,A -17.7727,B 24.8988,C -2.3219,E1 25.1562,E2 462.1798} C_DIS
LIN {X 71.0217,Y -17.9914,Z 79,A -20.3178,B 24.9002,C -2.3068,E1 25.1545,E2 464.746} C_DIS
LIN {X 70.1588,Y -21.1077,Z 79,A -22.5093,B 24.9,C -2.3087,E1 25.1528,E2 466.9203} C_DIS
LIN {X 69.2706,Y -23.8611,Z 79,A -24.8048,B 24.9007,C -2.3007,E1 25.1508,E2 469.2216} C_DIS
LIN {X 67.8656,Y -27.6038,Z 79,A -28.0182,B 24.9017,C -2.2887,E1 25.1476,E2 472.4457} C_DIS
LIN {X 66.9025,Y -29.8637,Z 79,A -30.3263,B 24.9032,C -2.2717,E1 25.145,E2 474.7811} C_DIS
LIN {X 64.8065,Y -34.1736,Z 79,A -33.4642,B 24.9026,C -2.2783,E1 25.1411,E2 477.8867} C_DIS
LIN {X 63.6422,Y -36.2966,Z 79,A -36.1453,B 24.905,C -2.2502,E1 25.1373,E2 480.6203} C_DIS
LIN {X 61.3694,Y -40.0206,Z 79,A -38.9884,B 24.9044,C -2.2569,E1 25.1332,E2 483.4332} C_DIS
LIN {X 59.5542,Y -42.6721,Z 79,A -41.4897,B 24.905,C -2.2504,E1 25.1292,E2 485.9378} C_DIS
LIN {X 57.1875,Y -45.7961,Z 79,A -45.1118,B 24.907,C -2.2264,E1 25.1229,E2 489.5994} C_DIS
LIN {X 54.9911,Y -48.4126,Z 79,A -47.7037,B 24.9074,C -2.2218,E1 25.1181,E2 492.1905} C_DIS
LIN {X 51.6374,Y -51.9744,Z 79,A -51.4006,B 24.9079,C -2.2162,E1 25.1109,E2 495.8849} C_DIS
LIN {X 47.6656,Y -55.6394,Z 79,A -55.7719,B 24.909,C -2.2025,E1 25.1018,E2 500.2712} C_DIS
LIN {X 43.6084,Y -58.8744,Z 79,A -59.2957,B 24.9085,C -2.2088,E1 25.094,E2 503.7671} C_DIS
LIN {X 40.5678,Y -61.0086,Z 79,A -62.2174,B 24.909,C -2.2026,E1 25.0873,E2 506.6936} C_DIS
LIN {X 36.1805,Y -63.7076,Z 79,A -66.386,B 24.9099,C -2.1913,E1 25.0773,E2 510.8758} C_DIS
LIN {X 33.6073,Y -65.1026,Z 79,A -68.8314,B 24.9106,C -2.1832,E1 25.0712,E2 513.3338} C_DIS
LIN {X 29.3903,Y -67.1114,Z 79,A -72.0236,B 24.91,C -2.1902,E1 25.0632,E2 516.5013} C_DIS
LIN {X 26.9482,Y -68.1288,Z 79,A -74.6967,B 24.9116,C -2.1708,E1 25.0561,E2 519.2141} C_DIS
LIN {X 22.6801,Y -69.6659,Z 79,A -77.6936,B 24.9108,C -2.1813,E1 25.0483,E2 522.1803} C_DIS
LIN {X 19.5864,Y -70.5992,Z 79,A -81.2287,B 24.9132,C -2.1516,E1 25.0386,E2 525.7801} C_DIS
LIN {X 15.5574,Y -71.5939,Z 79,A -83.1953,B 24.9106,C -2.1827,E1 25.0335,E2 527.6702} C_DIS
LIN {X 10.7925,Y -72.4666,Z 79,A -87.338,B 24.9117,C -2.1702,E1 25.022,E2 531.838} C_DIS
LIN {X 5.3806,Y -73.0682,Z 79,A -91.4069,B 24.9114,C -2.1729,E1 25.0108,E2 535.8979} C_DIS
LIN {X 1.4697,Y -73.25,Z 79,A -95.0088,B 24.9127,C -2.1578,E1 25.0006,E2 539.5349} C_DIS
LIN {X 1.4697,Y -73.25,Z 79,A -95.0088,B 24.9127,C -2.1578,E1 25.0006,E2 539.5349} C_DIS
Enddeposition()
LIN {X 0.4613,Y -72.3389,Z 79,A -94.732,B 24.9091,C -2.2015,E1 25.0017,E2 539.1542} C_DIS
Startdeposition()
$VEL.CP = VEL_PRINT
LIN {X 4.5123,Y -72.2129,Z 79,A -90.4971,B 24.9067,C -2.2296,E1 25.0137,E2 534.854} C_DIS
LIN {X 10.2469,Y -71.6236,Z 79,A -86.5052,B 24.9078,C -2.217,E1 25.0246,E2 530.8951} C_DIS
LIN {X 15.0579,Y -70.7695,Z 79,A -82.5997,B 24.9075,C -2.2211,E1 25.0354,E2 526.9843} C_DIS
LIN {X 19.3281,Y -69.7246,Z 79,A -79.4296,B 24.9079,C -2.2161,E1 25.0439,E2 523.8307} C_DIS
LIN {X 22.7229,Y -68.6933,Z 79,A -76.3011,B 24.9069,C -2.2281,E1 25.0523,E2 520.6796} C_DIS
LIN {X 27.1607,Y -67.0615,Z 79,A -72.8643,B 24.9072,C -2.2247,E1 25.0612,E2 517.2582} C_DIS
LIN {X 28.7676,Y -66.3881,Z 79,A -70.891,B 24.9056,C -2.2431,E1 25.0664,E2 515.2461} C_DIS
LIN {X 33.7537,Y -63.997,Z 79,A -66.4607,B 24.9049,C -2.2517,E1 25.0775,E2 510.8075} C_DIS
LIN {X 38.3253,Y -61.3686,Z 79,A -63.2931,B 24.9066,C -2.231,E1 25.0849,E2 507.6984} C_DIS
LIN {X 41.1562,Y -59.5074,Z 79,A -59.7445,B 24.9041,C -2.2605,E1 25.0933,E2 504.0918} C_DIS
LIN {X 44.4809,Y -57.0655,Z 79,A -56.5916,B 24.9038,C -2.2642,E1 25.1003,E2 500.9418} C_DIS
LIN {X 47.2782,Y -54.7712,Z 79,A -53.9153,B 24.9038,C -2.2652,E1 25.106,E2 498.2735} C_DIS
LIN {X 50.2256,Y -52.0797,Z 79,A -50.8277,B 24.9033,C -2.2705,E1 25.1123,E2 495.186} C_DIS
LIN {X 52.4554,Y -49.8329,Z 79,A -48.1483,B 24.9023,C -2.2815,E1 25.1175,E2 492.4919} C_DIS
LIN {X 54.6625,Y -47.4026,Z 79,A -45.7156,B 24.9022,C -2.2833,E1 25.122,E2 490.0659} C_DIS
LIN {X 58.0107,Y -43.2408,Z 79,A -41.2309,B 24.9006,C -2.3018,E1 25.1298,E2 485.5586} C_DIS
LIN {X 60.1864,Y -40.1582,Z 79,A -38.5403,B 24.9006,C -2.3014,E1 25.134,E2 482.8822} C_DIS
LIN {X 61.7996,Y -37.6264,Z 79,A -35.408,B 24.8981,C -2.3301,E1 25.1387,E2 479.698} C_DIS
LIN {X 63.621,Y -34.4572,Z 79,A -33.6737,B 24.9003,C -2.3047,E1 25.1409,E2 478.0328} C_DIS
LIN {X 65.2087,Y -31.349,Z 79,A -30.3072,B 24.8981,C -2.3303,E1 25.1452,E2 474.6238} C_DIS
LIN {X 66.7949,Y -27.8113,Z 79,A -27.1051,B 24.897,C -2.3434,E1 25.1487,E2 471.4082} C_DIS
LIN {X 68.201,Y -24.1578,Z 79,A -24.2083,B 24.8966,C -2.3469,E1 25.1514,E2 468.5194} C_DIS
LIN {X 69.2049,Y -21.112,Z 79,A -21.8763,B 24.8965,C -2.3487,E1 25.1534,E2 466.1964} C_DIS
LIN {X 70.0324,Y -18.1774,Z 79,A -19.5533,B 24.8961,C -2.3536,E1 25.1551,E2 463.8753} C_DIS
LIN {X 70.7603,Y -15.1,Z 79,A -16.4957,B 24.8939,C -2.3777,E1 25.1569,E2 460.7784} C_DIS
LIN {X 71.4327,Y -11.5097,Z 79,A -13.5521,B 24.893,C -2.3884,E1 25.1583,E2 457.827} C_DIS
LIN {X 72.1364,Y -5.5941,Z 79,A -9.144,B 24.8924,C -2.3942,E1 25.1595,E2 453.4311} C_DIS
LIN {X 72.3535,Y 0.107,Z 79,A -5.0753,B 24.8924,C -2.3954,E1 25.1598,E2 449.3838} C_DIS
LIN {X 72.2602,Y 3.6631,Z 79,A -2.1844,B 24.8913,C -2.4065,E1 25.1595,E2 446.4839} C_DIS
LIN {X 71.9716,Y 7.4185,Z 79,A 1.1117,B 24.8896,C -2.4251,E1 25.1586,E2 443.1635} C_DIS
LIN {X 71.1926,Y 12.9035,Z 79,A 5.3832,B 24.8887,C -2.4353,E1 25.1568,E2 438.893} C_DIS
LIN {X 70.4018,Y 16.6879,Z 79,A 8.3234,B 24.8882,C -2.4411,E1 25.155,E2 435.9561} C_DIS
LIN {X 69.689,Y 19.4538,Z 79,A 10.4074,B 24.888,C -2.4427,E1 25.1535,E2 433.8803} C_DIS
LIN {X 68.1453,Y 24.3166,Z 79,A 14.1138,B 24.8878,C -2.445,E1 25.1503,E2 430.1894} C_DIS
LIN {X 67.0513,Y 27.1857,Z 79,A 16.7424,B 24.8866,C -2.4577,E1 25.1476,E2 427.5455} C_DIS
LIN {X 66.0004,Y 29.6459,Z 79,A 19.8499,B 24.8834,C -2.4922,E1 25.144,E2 424.3731} C_DIS
LIN {X 64.2685,Y 33.2356,Z 79,A 22.1212,B 24.885,C -2.4753,E1 25.1412,E2 422.154} C_DIS
LIN {X 62.3813,Y 36.6543,Z 79,A 25.4056,B 24.8837,C -2.489,E1 25.1366,E2 418.8541} C_DIS
LIN {X 60.0014,Y 40.4325,Z 79,A 28.6752,B 24.8836,C -2.4904,E1 25.1316,E2 415.5975} C_DIS
LIN {X 58.35,Y 42.781,Z 79,A 31.5679,B 24.8814,C -2.5136,E1 25.1268,E2 412.664} C_DIS
LIN {X 56.3743,Y 45.3535,Z 79,A 33.1207,B 24.8835,C -2.4909,E1 25.1242,E2 411.1721} C_DIS
LIN {X 54.9904,Y 47.0213,Z 79,A 35.2393,B 24.8821,C -2.5062,E1 25.1204,E2 409.0272} C_DIS
LIN {X 52.8892,Y 49.3735,Z 79,A 37.9546,B 24.881,C -2.5178,E1 25.1152,E2 406.2963} C_DIS
LIN {X 50.2884,Y 52.0194,Z 79,A 40.6192,B 24.8811,C -2.5163,E1 25.11,E2 403.6466} C_DIS
LIN {X 46.5284,Y 55.4092,Z 79,A 44.3126,B 24.8812,C -2.5153,E1 25.1023,E2 399.9701} C_DIS
LIN {X 44.8487,Y 56.7761,Z 79,A 46.311,B 24.8802,C -2.5263,E1 25.0979,E2 397.9532} C_DIS
LIN {X 40.7824,Y 59.7645,Z 79,A 50.0456,B 24.8802,C -2.5259,E1 25.0895,E2 394.2327} C_DIS
LIN {X 38.7292,Y 61.1159,Z 79,A 52.2919,B 24.8792,C -2.5371,E1 25.0841,E2 391.9673} C_DIS
LIN {X 36.0127,Y 62.7536,Z 79,A 54.729,B 24.879,C -2.5387,E1 25.0783,E2 389.5338} C_DIS
LIN {X 32.3156,Y 64.7354,Z 79,A 57.8787,B 24.879,C -2.5383,E1 25.0705,E2 386.3938} C_DIS
LIN {X 29.0777,Y 66.2529,Z 79,A 61.1012,B 24.8777,C -2.552,E1 25.0623,E2 383.1469} C_DIS
LIN {X 24.5967,Y 68.0439,Z 79,A 64.6855,B 24.878,C -2.5493,E1 25.053,E2 379.5768} C_DIS
LIN {X 22.2123,Y 68.8589,Z 79,A 67.2082,B 24.8765,C -2.5649,E1 25.0462,E2 377.0217} C_DIS
LIN {X 17.8404,Y 70.119,Z 79,A 70.3139,B 24.8775,C -2.5541,E1 25.0379,E2 373.9469} C_DIS
LIN {X 14.8104,Y 70.8213,Z 79,A 72.7535,B 24.8775,C -2.5547,E1 25.0312,E2 371.509} C_DIS
LIN {X 11.4545,Y 71.4406,Z 79,A 76.0537,B 24.8759,C -2.5712,E1 25.0221,E2 368.1729} C_DIS
LIN {X 7.5173,Y 71.9612,Z 79,A 78.532,B 24.8775,C -2.5544,E1 25.0153,E2 365.7364} C_DIS
LIN {X 3.6806,Y 72.2598,Z 79,A 81.6711,B 24.8773,C -2.5568,E1 25.0065,E2 362.5929} C_DIS
LIN {X -0.9438,Y 72.3477,Z 79,A 85.3112,B 24.8773,C -2.5556,E1 24.9964,E2 358.9561} C_DIS
LIN {X -4.012,Y 72.2415,Z 79,A 88.5169,B 24.8756,C -2.5744,E1 24.9873,E2 355.7046} C_DIS
LIN {X -7.6378,Y 71.9486,Z 79,A 90.4478,B 24.878,C -2.549,E1 24.9821,E2 353.8333} C_DIS
LIN {X -12.682,Y 71.2328,Z 79,A 94.662,B 24.8779,C -2.5507,E1 24.9705,E2 349.6113} C_DIS
LIN {X -15.8193,Y 70.6035,Z 79,A 97.3489,B 24.8777,C -2.5523,E1 24.9631,E2 346.9173} C_DIS
LIN {X -20.221,Y 69.4703,Z 79,A 100.9084,B 24.8782,C -2.5477,E1 24.9535,E2 343.3634} C_DIS
LIN {X -23.57,Y 68.4073,Z 79,A 103.6516,B 24.8786,C -2.5434,E1 24.9463,E2 340.6253} C_DIS
LIN {X -26.4743,Y 67.3353,Z 79,A 106.8465,B 24.8771,C -2.5583,E1 24.9379,E2 337.3879} C_DIS
LIN {X -29.8418,Y 65.9122,Z 79,A 108.994,B 24.8793,C -2.5359,E1 24.9325,E2 335.2887} C_DIS
LIN {X -33.3587,Y 64.2041,Z 79,A 112.1028,B 24.8797,C -2.5313,E1 24.9247,E2 332.1827} C_DIS
LIN {X -37.3334,Y 61.9777,Z 79,A 115.3271,B 24.8812,C -2.5159,E1 24.917,E2 328.9856} C_DIS
LIN {X -39.7166,Y 60.4776,Z 79,A 117.5085,B 24.8817,C -2.5106,E1 24.9119,E2 326.8099} C_DIS
LIN {X -43.5817,Y 57.7545,Z 79,A 121.5954,B 24.8817,C -2.5111,E1 24.9026,E2 322.7076} C_DIS
LIN {X -48.1097,Y 54.041,Z 79,A 125.9266,B 24.8833,C -2.4938,E1 24.8933,E2 318.4012} C_DIS
LIN {X -51.7917,Y 50.5247,Z 79,A 130.1571,B 24.8837,C -2.4889,E1 24.8848,E2 314.1648} C_DIS
LIN {X -55.5108,Y 46.4062,Z 79,A 134.7774,B 24.8843,C -2.4831,E1 24.8762,E2 309.5377} C_DIS
LIN {X -58.1826,Y 43.0096,Z 79,A 138.1466,B 24.8852,C -2.4728,E1 24.8705,E2 306.1769} C_DIS
LIN {X -59.7132,Y 40.8581,Z 79,A 141.2097,B 24.8837,C -2.4895,E1 24.8655,E2 303.0588} C_DIS
LIN {X -61.743,Y 37.7195,Z 79,A 143.1252,B 24.8867,C -2.4573,E1 24.8628,E2 301.2106} C_DIS
LIN {X -62.6863,Y 36.1299,Z 79,A 145.5666,B 24.885,C -2.4754,E1 24.8594,E2 298.7131} C_DIS
LIN {X -64.3658,Y 33.0453,Z 79,A 147.3693,B 24.8878,C -2.445,E1 24.8571,E2 296.9734} C_DIS
LIN {X -65.5437,Y 30.6425,Z 79,A 149.7173,B 24.8879,C -2.4439,E1 24.8542,E2 294.6152} C_DIS
LIN {X -66.8311,Y 27.7254,Z 79,A 152.368,B 24.8883,C -2.4392,E1 24.8513,E2 291.9612} C_DIS
LIN {X -67.9798,Y 24.7725,Z 79,A 155.3322,B 24.8881,C -2.4419,E1 24.8484,E2 288.9738} C_DIS
LIN {X -69.4934,Y 20.1442,Z 79,A 158.8663,B 24.8899,C -2.4227,E1 24.8455,E2 285.4653} C_DIS
LIN {X -70.5899,Y 15.8798,Z 79,A 162.2821,B 24.891,C -2.4101,E1 24.8433,E2 282.0594} C_DIS
LIN {X -71.2233,Y 12.7347,Z 79,A 164.8016,B 24.8918,C -2.4017,E1 24.842,E2 279.5453} C_DIS
LIN {X -71.7128,Y 9.6073,Z 79,A 167.6538,B 24.8918,C -2.4015,E1 24.8409,E2 276.6764} C_DIS
LIN {X -72.0743,Y 6.3497,Z 79,A 170.2243,B 24.8926,C -2.3927,E1 24.8402,E2 274.1116} C_DIS
LIN {X -72.2687,Y 3.5106,Z 79,A 172.2424,B 24.8937,C -2.3802,E1 24.8399,E2 272.1112} C_DIS
LIN {X -72.3517,Y 0.3975,Z 79,A 174.56,B 24.8947,C -2.3691,E1 24.8398,E2 269.8063} C_DIS
LIN {X -72.3072,Y -2.5975,Z 79,A 177.1343,B 24.8949,C -2.3661,E1 24.84,E2 267.2235} C_DIS
LIN {X -72.0925,Y -6.1438,Z 79,A 179.7166,B 24.8962,C -2.352,E1 24.8405,E2 264.6593} C_DIS
LIN {X -71.8219,Y -8.756,Z 79,A -177.9683,B 24.8963,C -2.3508,E1 24.8412,E2 262.3333} C_DIS
LIN {X -71.3976,Y -11.7198,Z 79,A -175.4192,B 24.8966,C -2.3475,E1 24.8423,E2 259.7769} C_DIS
LIN {X -70.7083,Y -15.3387,Z 79,A -172.6857,B 24.8978,C -2.3344,E1 24.8438,E2 257.0586} C_DIS
LIN {X -70.0428,Y -18.1372,Z 79,A -170.3712,B 24.8983,C -2.3283,E1 24.8454,E2 254.745} C_DIS
LIN {X -68.9438,Y -21.9476,Z 79,A -167.2286,B 24.8991,C -2.319,E1 24.8479,E2 251.6065} C_DIS
LIN {X -67.245,Y -26.704,Z 79,A -163.3042,B 24.9003,C -2.3057,E1 24.8517,E2 247.6919} C_DIS
LIN {X -65.3717,Y -31.0098,Z 79,A -159.764,B 24.9015,C -2.2911,E1 24.8557,E2 244.167} C_DIS
LIN {X -63.7576,Y -34.2054,Z 79,A -156.1017,B 24.9005,C -2.3025,E1 24.8605,E2 240.4578} C_DIS
LIN {X -61.6956,Y -37.7974,Z 79,A -153.2596,B 24.9022,C -2.2838,E1 24.8645,E2 237.6459} C_DIS
LIN {X -59.8915,Y -40.5949,Z 79,A -150.6563,B 24.9028,C -2.2763,E1 24.8685,E2 235.0473} C_DIS
LIN {X -57.4018,Y -44.0453,Z 79,A -147.4286,B 24.9038,C -2.2648,E1 24.8738,E2 231.8313} C_DIS
LIN {X -55.6752,Y -46.2083,Z 79,A -145.046,B 24.9038,C -2.2642,E1 24.878,E2 229.4392} C_DIS
LIN {X -52.9275,Y -49.3327,Z 79,A -142.0858,B 24.9051,C -2.249,E1 24.8835,E2 226.502} C_DIS
LIN {X -50.1589,Y -52.1443,Z 79,A -138.5625,B 24.9049,C -2.2519,E1 24.8905,E2 222.9568} C_DIS
LIN {X -47.8281,Y -54.2909,Z 79,A -136.1128,B 24.9054,C -2.2456,E1 24.8956,E2 220.5125} C_DIS
LIN {X -45.5631,Y -56.2044,Z 79,A -133.2609,B 24.9047,C -2.2535,E1 24.9018,E2 217.631} C_DIS
LIN {X -41.579,Y -59.2135,Z 79,A -129.7137,B 24.9061,C -2.2369,E1 24.9097,E2 214.1109} C_DIS
LIN {X -38.7668,Y -61.0918,Z 79,A -127.0394,B 24.9065,C -2.2326,E1 24.916,E2 211.438} C_DIS
LIN {X -34.9632,Y -63.3454,Z 79,A -123.7948,B 24.9074,C -2.2214,E1 24.9238,E2 208.2104} C_DIS
LIN {X -31.812,Y -64.9837,Z 79,A -120.6932,B 24.9071,C -2.2251,E1 24.9315,E2 205.0917} C_DIS
LIN {X -29.0536,Y -66.2634,Z 79,A -118.3824,B 24.9075,C -2.22,E1 24.9374,E2 202.7874} C_DIS
LIN {X -27.0123,Y -67.1219,Z 79,A -116.4553,B 24.9073,C -2.2226,E1 24.9424,E2 200.8497} C_DIS
LIN {X -22.2603,Y -68.8434,Z 79,A -112.5308,B 24.9078,C -2.2173,E1 24.9528,E2 196.9303} C_DIS
LIN {X -19.2718,Y -69.7402,Z 79,A -110.0727,B 24.9079,C -2.2154,E1 24.9593,E2 194.4729} C_DIS
LIN {X -16.1553,Y -70.5263,Z 79,A -107.6199,B 24.9082,C -2.2117,E1 24.966,E2 192.0254} C_DIS
LIN {X -11.1667,Y -71.486,Z 79,A -103.8622,B 24.9089,C -2.2035,E1 24.9763,E2 188.2833} C_DIS
LIN {X -6.3728,Y -72.0721,Z 79,A -100.0957,B 24.9091,C -2.2013,E1 24.9867,E2 184.5193} C_DIS
LIN {X -1.7002,Y -72.3338,Z 79,A -96.199,B 24.9087,C -2.2065,E1 24.9976,E2 180.6093} C_DIS
LIN {X 0.4613,Y -72.3389,Z 79,A -94.7302,B 24.9092,C -2.2007,E1 25.0017,E2 179.1542} C_DIS
Enddeposition()
LIN {X 0.4613,Y -72.3389,Z 79,A -94.7302,B 24.9092,C -2.2007,E1 25.0017,E2 179.1542} C_DIS
Startdeposition()
$VEL.CP = VEL_PRINT
LIN {X -1.2546,Y -71.43,Z 79,A -96.5848,B 24.9089,C -2.2038,E1 24.9965,E2 181.0016} C_DIS
LIN {X -4.3415,Y -71.3095,Z 79,A -99.7796,B 24.9104,C -2.1856,E1 24.9875,E2 184.2406} C_DIS
LIN {X -8.498,Y -70.934,Z 79,A -102.6767,B 24.9094,C -2.1971,E1 24.9795,E2 187.1119} C_DIS
LIN {X -11.5012,Y -70.5097,Z 79,A -105.2397,B 24.9097,C -2.1945,E1 24.9724,E2 189.6834} C_DIS
LIN {X -14.9242,Y -69.8654,Z 79,A -107.8781,B 24.9093,C -2.1994,E1 24.9652,E2 192.313} C_DIS
LIN {X -17.7295,Y -69.2061,Z 79,A -110.054,B 24.9089,C -2.204,E1 24.9593,E2 194.481} C_DIS
LIN {X -20.3935,Y -68.4684,Z 79,A -112.418,B 24.9091,C -2.2019,E1 24.953,E2 196.854} C_DIS
LIN {X -23.2897,Y -67.5392,Z 79,A -115.0218,B 24.9092,C -2.1998,E1 24.946,E2 199.4677} C_DIS
LIN {X -26.9327,Y -66.1698,Z 79,A -118.8695,B 24.9104,C -2.1855,E1 24.9359,E2 203.3579} C_DIS
LIN {X -30.4947,Y -64.6067,Z 79,A -121.1598,B 24.9085,C -2.2086,E1 24.9303,E2 205.5987} C_DIS
LIN {X -33.3813,Y -63.1626,Z 79,A -123.7426,B 24.9082,C -2.212,E1 24.9238,E2 208.1804} C_DIS
LIN {X -35.326,Y -62.0965,Z 79,A -125.4711,B 24.9079,C -2.2156,E1 24.9197,E2 209.9054} C_DIS
LIN {X -37.616,Y -60.7365,Z 79,A -127.5628,B 24.9076,C -2.2198,E1 24.9147,E2 211.9936} C_DIS
LIN {X -40.0918,Y -59.1309,Z 79,A -129.8771,B 24.9072,C -2.2247,E1 24.9093,E2 214.3038} C_DIS
LIN {X -43.1216,Y -56.9597,Z 79,A -133.1168,B 24.9072,C -2.2239,E1 24.902,E2 217.5568} C_DIS
LIN {X -45.8105,Y -54.8201,Z 79,A -135.7629,B 24.9066,C -2.2315,E1 24.8962,E2 220.1948} C_DIS
LIN {X -48.1326,Y -52.7931,Z 79,A -138.2325,B 24.9062,C -2.2364,E1 24.8911,E2 222.6626} C_DIS
LIN {X -50.3755,Y -50.6574,Z 79,A -141.0311,B 24.9064,C -2.2343,E1 24.8855,E2 225.4779} C_DIS
LIN {X -53.1737,Y -47.7114,Z 79,A -144.0084,B 24.9052,C -2.2478,E1 24.8799,E2 228.4361} C_DIS
LIN {X -55.2396,Y -45.3053,Z 79,A -146.6793,B 24.905,C -2.2507,E1 24.8751,E2 231.1123} C_DIS
LIN {X -56.7658,Y -43.3767,Z 79,A -149.3975,B 24.906,C -2.2387,E1 24.8704,E2 233.872} C_DIS
LIN {X -58.9386,Y -40.3757,Z 79,A -151.6682,B 24.904,C -2.2617,E1 24.8668,E2 236.0992} C_DIS
LIN {X -60.7426,Y -37.6062,Z 79,A -154.1179,B 24.9031,C -2.273,E1 24.8632,E2 238.5343} C_DIS
LIN {X -62.1677,Y -35.2018,Z 79,A -156.5518,B 24.9029,C -2.2746,E1 24.8598,E2 240.977} C_DIS
LIN {X -63.7176,Y -32.3099,Z 79,A -159.0376,B 24.902,C -2.285,E1 24.8566,E2 243.4513} C_DIS
LIN {X -64.7012,Y -30.2916,Z 79,A -161.0261,B 24.902,C -2.2858,E1 24.8542,E2 245.4486} C_DIS
LIN {X -65.8718,Y -27.6535,Z 79,A -163.0658,B 24.9009,C -2.2984,E1 24.8519,E2 247.4695} C_DIS
LIN {X -66.9262,Y -24.9958,Z 79,A -165.8803,B 24.9013,C -2.2936,E1 24.8491,E2 250.3114} C_DIS
LIN {X -68.546,Y -20.1318,Z 79,A -169.6924,B 24.8997,C -2.3123,E1 24.8459,E2 254.1006} C_DIS
LIN {X -69.3016,Y -17.3575,Z 79,A -172.102,B 24.8993,C -2.3169,E1 24.8442,E2 256.5132} C_DIS
LIN {X -69.9429,Y -14.5545,Z 79,A -174.0856,B 24.898,C -2.331,E1 24.843,E2 258.4747} C_DIS
LIN {X -70.4066,Y -12.1177,Z 79,A -176.3363,B 24.898,C -2.3315,E1 24.8419,E2 260.7377} C_DIS
LIN {X -70.822,Y -9.3857,Z 79,A -178.5903,B 24.8975,C -2.3375,E1 24.841,E2 262.9907} C_DIS
LIN {X -71.1809,Y -6.104,Z 79,A 178.9912,B 24.8963,C -2.3508,E1 24.8403,E2 265.392} C_DIS
LIN {X -71.312,Y -4.3056,Z 79,A 177.2569,B 24.8965,C -2.3491,E1 24.84,E2 267.1407} C_DIS
LIN {X -71.4285,Y -1.3359,Z 79,A 174.945,B 24.8956,C -2.3582,E1 24.8398,E2 269.4449} C_DIS
LIN {X -71.4219,Y 1.6929,Z 79,A 172.4319,B 24.8951,C -2.3641,E1 24.8398,E2 271.9591} C_DIS
LIN {X -71.2988,Y 4.5154,Z 79,A 170.0374,B 24.8947,C -2.3685,E1 24.8402,E2 274.3574} C_DIS
LIN {X -71.0623,Y 7.3464,Z 79,A 167.9555,B 24.8937,C -2.38,E1 24.8408,E2 276.4243} C_DIS
LIN {X -70.703,Y 10.2434,Z 79,A 165.6359,B 24.893,C -2.3879,E1 24.8416,E2 278.7389} C_DIS
LIN {X -70.2813,Y 12.8209,Z 79,A 163.4372,B 24.8926,C -2.3923,E1 24.8427,E2 280.9402} C_DIS
LIN {X -69.6964,Y 15.6962,Z 79,A 160.9511,B 24.8922,C -2.3968,E1 24.8441,E2 283.4303} C_DIS
LIN {X -68.825,Y 19.1583,Z 79,A 158.1764,B 24.8912,C -2.4076,E1 24.8461,E2 286.1952} C_DIS
LIN {X -68.2383,Y 21.1504,Z 79,A 156.2336,B 24.8912,C -2.4068,E1 24.8477,E2 288.1511} C_DIS
LIN {X -66.9764,Y 24.8624,Z 79,A 153.3589,B 24.8899,C -2.4222,E1 24.8504,E2 291.0053} C_DIS
LIN {X -65.9005,Y 27.5856,Z 79,A 151.029,B 24.8892,C -2.4297,E1 24.8528,E2 293.3303} C_DIS
LIN {X -64.6957,Y 30.3035,Z 79,A 148.5849,B 24.8887,C -2.4355,E1 24.8556,E2 295.774} C_DIS
LIN {X -63.3538,Y 33.0182,Z 79,A 146.064,B 24.8882,C -2.4405,E1 24.8588,E2 298.2963} C_DIS
LIN {X -61.5039,Y 36.3466,Z 79,A 143.2496,B 24.8869,C -2.4545,E1 24.8626,E2 301.092} C_DIS
LIN {X -60.078,Y 38.6581,Z 79,A 140.7921,B 24.8869,C -2.4545,E1 24.8663,E2 303.5622} C_DIS
LIN {X -58.3349,Y 41.2426,Z 79,A 138.3246,B 24.8862,C -2.462,E1 24.8702,E2 306.0239} C_DIS
LIN {X -56.8723,Y 43.2379,Z 79,A 136.1023,B 24.8862,C -2.462,E1 24.874,E2 308.2568} C_DIS
LIN {X -54.8424,Y 45.7837,Z 79,A 133.0367,B 24.8865,C -2.4588,E1 24.8795,E2 311.3443} C_DIS
LIN {X -51.6637,Y 49.3435,Z 79,A 129.8091,B 24.8844,C -2.4814,E1 24.8855,E2 314.532} C_DIS
LIN {X -49.1753,Y 51.8238,Z 79,A 126.9739,B 24.8838,C -2.4877,E1 24.8911,E2 317.3642} C_DIS
LIN {X -47.456,Y 53.4023,Z 79,A 124.712,B 24.8843,C -2.4832,E1 24.8959,E2 319.6458} C_DIS
LIN {X -44.3914,Y 55.9752,Z 79,A 121.8548,B 24.8829,C -2.498,E1 24.902,E2 322.4785} C_DIS
LIN {X -41.8264,Y 57.9183,Z 79,A 118.8924,B 24.8832,C -2.4946,E1 24.9087,E2 325.4594} C_DIS
LIN {X -39.09,Y 59.7985,Z 79,A 116.5397,B 24.882,C -2.5068,E1 24.9142,E2 327.7909} C_DIS
LIN {X -34.1691,Y 62.7399,Z 79,A 112.0732,B 24.881,C -2.5179,E1 24.9249,E2 332.2442} C_DIS
LIN {X -31.5592,Y 64.0926,Z 79,A 109.6806,B 24.8807,C -2.5209,E1 24.9309,E2 334.6361} C_DIS
LIN {X -28.9534,Y 65.3122,Z 79,A 107.504,B 24.8801,C -2.5274,E1 24.9364,E2 336.8026} C_DIS
LIN {X -26.3307,Y 66.412,Z 79,A 105.0923,B 24.8801,C -2.5274,E1 24.9426,E2 339.2195} C_DIS
LIN {X -23.6633,Y 67.4081,Z 79,A 102.7775,B 24.8799,C -2.5296,E1 24.9487,E2 341.5339} C_DIS
LIN {X -20.8552,Y 68.3297,Z 79,A 99.9921,B 24.8806,C -2.5226,E1 24.9562,E2 344.341} C_DIS
LIN {X -17.125,Y 69.3584,Z 79,A 97.2647,B 24.8794,C -2.5345,E1 24.9635,E2 347.0439} C_DIS
LIN {X -14.1027,Y 70.0357,Z 79,A 94.7228,B 24.8794,C -2.5353,E1 24.9704,E2 349.5872} C_DIS
LIN {X -11.948,Y 70.435,Z 79,A 92.6943,B 24.8798,C -2.5301,E1 24.976,E2 351.6301} C_DIS
LIN {X -7.9775,Y 70.9949,Z 79,A 89.485,B 24.8796,C -2.5321,E1 24.9849,E2 354.8368} C_DIS
LIN {X -4.1172,Y 71.3224,Z 79,A 86.7493,B 24.8787,C -2.5424,E1 24.9925,E2 357.549} C_DIS
LIN {X -1.202,Y 71.4309,Z 79,A 84.6788,B 24.878,C -2.5497,E1 24.9982,E2 359.6024} C_DIS
LIN {X 0.9611,Y 71.435,Z 79,A 82.2631,B 24.8795,C -2.5332,E1 25.005,E2 362.057} C_DIS
LIN {X 4.9783,Y 71.2675,Z 79,A 79.3768,B 24.8787,C -2.5417,E1 25.013,E2 364.9222} C_DIS
LIN {X 7.8794,Y 71.0064,Z 79,A 77.2835,B 24.8782,C -2.5474,E1 25.0188,E2 367.0005} C_DIS
LIN {X 10.1726,Y 70.7131,Z 79,A 75.0657,B 24.8791,C -2.5379,E1 25.025,E2 369.2391} C_DIS
LIN {X 13.4925,Y 70.1553,Z 79,A 72.4927,B 24.8789,C -2.5401,E1 25.0321,E2 371.804} C_DIS
LIN {X 16.525,Y 69.5048,Z 79,A 69.954,B 24.8791,C -2.5375,E1 25.039,E2 374.3455} C_DIS
LIN {X 19.5659,Y 68.7095,Z 79,A 67.7625,B 24.8785,C -2.5443,E1 25.0448,E2 376.5173} C_DIS
LIN {X 21.8608,Y 68.0142,Z 79,A 65.6714,B 24.879,C -2.5386,E1 25.0504,E2 378.6183} C_DIS
LIN {X 23.877,Y 67.3331,Z 79,A 63.0076,B 24.8815,C -2.5126,E1 25.0576,E2 381.3382} C_DIS
LIN {X 27.4161,Y 65.9719,Z 79,A 60.7288,B 24.8799,C -2.529,E1 25.0634,E2 383.5729} C_DIS
LIN {X 30.4123,Y 64.6451,Z 79,A 58.1838,B 24.88,C -2.5282,E1 25.0698,E2 386.1134} C_DIS
LIN {X 33.5883,Y 63.0535,Z 79,A 55.4596,B 24.88,C -2.5279,E1 25.0766,E2 388.831} C_DIS
LIN {X 35.8836,Y 61.7761,Z 79,A 53.208,B 24.8807,C -2.5211,E1 25.0821,E2 391.0919} C_DIS
LIN {X 38.346,Y 60.2783,Z 79,A 50.9838,B 24.8808,C -2.5199,E1 25.0873,E2 393.3118} C_DIS
LIN {X 40.6058,Y 58.7794,Z 79,A 48.6485,B 24.8815,C -2.5121,E1 25.0927,E2 395.6576} C_DIS
LIN {X 43.244,Y 56.8677,Z 79,A 46.1284,B 24.8817,C -2.5101,E1 25.0984,E2 398.1735} C_DIS
LIN {X 45.7353,Y 54.8826,Z 79,A 43.6435,B 24.882,C -2.5072,E1 25.1037,E2 400.6558} C_DIS
LIN {X 48.2897,Y 52.649,Z 79,A 40.9931,B 24.8823,C -2.5038,E1 25.1093,E2 403.3037} C_DIS
LIN {X 50.0397,Y 50.9891,Z 79,A 39.1213,B 24.8825,C -2.5015,E1 25.113,E2 405.1732} C_DIS
LIN {X 51.9061,Y 49.0877,Z 79,A 36.9097,B 24.8832,C -2.4949,E1 25.1173,E2 407.3909} C_DIS
LIN {X 53.9537,Y 46.828,Z 79,A 34.4281,B 24.8838,C -2.4884,E1 25.1219,E2 409.8767} C_DIS
LIN {X 55.8733,Y 44.5204,Z 79,A 32.4115,B 24.8833,C -2.4935,E1 25.1255,E2 411.8718} C_DIS
LIN {X 57.2454,Y 42.7413,Z 79,A 30.2162,B 24.8847,C -2.4784,E1 25.1292,E2 414.0925} C_DIS
LIN {X 58.9183,Y 40.4057,Z 79,A 28.1936,B 24.8845,C -2.4804,E1 25.1324,E2 416.1005} C_DIS
LIN {X 60.012,Y 38.7608,Z 79,A 26.151,B 24.8861,C -2.4638,E1 25.1356,E2 418.1723} C_DIS
LIN {X 62.4814,Y 34.6401,Z 79,A 22.5414,B 24.8864,C -2.4603,E1 25.1406,E2 421.7714} C_DIS
LIN {X 63.7986,Y 32.1514,Z 79,A 19.7272,B 24.8884,C -2.4387,E1 25.1443,E2 424.6216} C_DIS
LIN {X 65.7242,Y 28.004,Z 79,A 16.684,B 24.8877,C -2.4457,E1 25.1477,E2 427.6317} C_DIS
LIN {X 66.7265,Y 25.5233,Z 79,A 14.544,B 24.8883,C -2.4397,E1 25.1499,E2 429.7741} C_DIS
LIN {X 67.8684,Y 22.3116,Z 79,A 11.7733,B 24.8891,C -2.4306,E1 25.1524,E2 432.5506} C_DIS
LIN {X 68.8637,Y 19.02,Z 79,A 9.168,B 24.8895,C -2.4267,E1 25.1544,E2 435.1504} C_DIS
LIN {X 69.5998,Y 16.1145,Z 79,A 6.094,B 24.8919,C -2.4006,E1 25.1564,E2 438.2682} C_DIS
LIN {X 70.5204,Y 11.4371,Z 79,A 2.8432,B 24.8915,C -2.4048,E1 25.158,E2 441.4899} C_DIS
LIN {X 70.8924,Y 8.8426,Z 79,A 0.4897,B 24.8927,C -2.3912,E1 25.1589,E2 443.8618} C_DIS
LIN {X 71.3092,Y 4.3556,Z 79,A -2.8358,B 24.893,C -2.3879,E1 25.1596,E2 447.1753} C_DIS
LIN {X 71.4306,Y 1.2214,Z 79,A -5.3257,B 24.8936,C -2.3807,E1 25.1598,E2 449.6674} C_DIS
LIN {X 71.3329,Y -3.9273,Z 79,A -9.3616,B 24.8946,C -2.3703,E1 25.1594,E2 453.704} C_DIS
LIN {X 70.8283,Y -9.3375,Z 79,A -13.7532,B 24.8959,C -2.3554,E1 25.1582,E2 458.1046} C_DIS
LIN {X 70.3656,Y -12.3523,Z 79,A -16.3336,B 24.8969,C -2.3439,E1 25.157,E2 460.6972} C_DIS
LIN {X 69.6624,Y -15.8437,Z 79,A -18.9497,B 24.8971,C -2.3417,E1 25.1555,E2 463.3033} C_DIS
LIN {X 68.9519,Y -18.6936,Z 79,A -21.2179,B 24.8975,C -2.3368,E1 25.1539,E2 465.5699} C_DIS
LIN {X 68.1698,Y -21.3715,Z 79,A -23.3988,B 24.898,C -2.3314,E1 25.1521,E2 467.7511} C_DIS
LIN {X 67.4469,Y -23.5527,Z 79,A -26.1408,B 24.9007,C -2.3005,E1 25.1495,E2 470.5507} C_DIS
LIN {X 66.1783,Y -26.9118,Z 79,A -28.0735,B 24.8992,C -2.3183,E1 25.1476,E2 472.4306} C_DIS
LIN {X 65.4471,Y -28.6443,Z 79,A -29.9944,B 24.9006,C -2.3022,E1 25.1454,E2 474.3792} C_DIS
LIN {X 63.8378,Y -32.0732,Z 79,A -32.7294,B 24.9006,C -2.3017,E1 25.1421,E2 477.1006} C_DIS
LIN {X 62.4953,Y -34.6151,Z 79,A -35.3574,B 24.902,C -2.286,E1 25.1386,E2 479.752} C_DIS
LIN {X 60.3811,Y -38.1849,Z 79,A -38.4101,B 24.9021,C -2.2842,E1 25.1341,E2 482.7933} C_DIS
LIN {X 58.7919,Y -40.5879,Z 79,A -40.5646,B 24.9023,C -2.2822,E1 25.1308,E2 484.9418} C_DIS
LIN {X 57.3303,Y -42.6282,Z 79,A -42.837,B 24.9034,C -2.2696,E1 25.127,E2 487.2332} C_DIS
LIN {X 55.1118,Y -45.4595,Z 79,A -45.494,B 24.9034,C -2.2684,E1 25.1224,E2 489.8807} C_DIS
LIN {X 52.9491,Y -47.9622,Z 79,A -47.9126,B 24.9034,C -2.2681,E1 25.1179,E2 492.2889} C_DIS
LIN {X 51.0493,Y -49.9788,Z 79,A -50.6416,B 24.9051,C -2.2487,E1 25.1126,E2 495.0522} C_DIS
LIN {X 48.3139,Y -52.6268,Z 79,A -53.4202,B 24.9051,C -2.2491,E1 25.107,E2 497.8184} C_DIS
LIN {X 45.9078,Y -54.7392,Z 79,A -55.9623,B 24.9055,C -2.244,E1 25.1016,E2 500.3625} C_DIS
LIN {X 44.1221,Y -56.1881,Z 79,A -57.8876,B 24.9061,C -2.2378,E1 25.0973,E2 502.2953} C_DIS
LIN {X 41.1733,Y -58.3843,Z 79,A -60.7397,B 24.9063,C -2.2344,E1 25.0909,E2 505.1455} C_DIS
LIN {X 38.6645,Y -60.0739,Z 79,A -62.9888,B 24.9063,C -2.2345,E1 25.0857,E2 507.3868} C_DIS
LIN {X 35.4116,Y -62.0474,Z 79,A -66.2056,B 24.9072,C -2.2245,E1 25.0779,E2 510.6175} C_DIS
LIN {X 32.3313,Y -63.7066,Z 79,A -69.1035,B 24.9078,C -2.2173,E1 25.0707,E2 513.5242} C_DIS
LIN {X 28.1449,Y -65.6648,Z 79,A -72.4177,B 24.9074,C -2.2222,E1 25.0624,E2 516.8186} C_DIS
LIN {X 25.6129,Y -66.6926,Z 79,A -74.8304,B 24.9081,C -2.2132,E1 25.0561,E2 519.2471} C_DIS
LIN {X 22.9987,Y -67.638,Z 79,A -76.9892,B 24.9081,C -2.2123,E1 25.0504,E2 521.4038} C_DIS
LIN {X 20.2304,Y -68.5168,Z 79,A -79.2186,B 24.9081,C -2.2123,E1 25.0444,E2 523.6293} C_DIS
LIN {X 17.6877,Y -69.2168,Z 79,A -82.0234,B 24.9099,C -2.192,E1 25.0367,E2 526.4777} C_DIS
LIN {X 12.8689,Y -70.2727,Z 79,A -85.4723,B 24.9091,C -2.2018,E1 25.0274,E2 529.8992} C_DIS
LIN {X 10.1763,Y -70.7126,Z 79,A -88.4352,B 24.9108,C -2.1804,E1 25.0191,E2 532.9102} C_DIS
LIN {X 6.5669,Y -71.1385,Z 79,A -90.5902,B 24.9094,C -2.1982,E1 25.0132,E2 535.0216} C_DIS
LIN {X 1.7792,Y -71.42,Z 79,A -94.3884,B 24.9094,C -2.198,E1 25.0026,E2 538.8191} C_DIS
LIN {X 1.7792,Y -71.42,Z 79,A -94.3884,B 24.9094,C -2.198,E1 25.0026,E2 538.8191} C_DIS
Enddeposition()
LIN {X 0.4365,Y -70.5262,Z 79,A -94.5503,B 24.9061,C -2.2369,E1 25.0024,E2 538.8885} C_DIS
Startdeposition()
$VEL.CP = VEL_PRINT
LIN {X 3.2195,Y -70.4558,Z 79,A -92.2942,B 24.9061,C -2.2375,E1 25.0087,E2 536.6316} C_DIS
LIN {X 5.4004,Y -70.3224,Z 79,A -90.3453,B 24.9056,C -2.2428,E1 25.0142,E2 534.671} C_DIS
LIN {X 8.3902,Y -70.0285,Z 79,A -88.0828,B 24.9059,C -2.2396,E1 25.0204,E2 532.4177} C_DIS
LIN {X 10.5638,Y -69.7338,Z 79,A -86.1302,B 24.9054,C -2.2452,E1 25.0259,E2 530.4534} C_DIS
LIN {X 13.5233,Y -69.2207,Z 79,A -83.8683,B 24.9057,C -2.2425,E1 25.032,E2 528.2005} C_DIS
LIN {X 16.0395,Y -68.6813,Z 79,A -81.6722,B 24.9053,C -2.2472,E1 25.038,E2 525.9962} C_DIS
LIN {X 18.7965,Y -67.9795,Z 79,A -79.2277,B 24.9048,C -2.2531,E1 25.0447,E2 523.5415} C_DIS
LIN {X 21.5023,Y -67.1718,Z 79,A -77.0108,B 24.9048,C -2.2537,E1 25.0506,E2 521.3272} C_DIS
LIN {X 24.3556,Y -66.1906,Z 79,A -74.744,B 24.9048,C -2.2519,E1 25.0565,E2 519.0692} C_DIS
LIN {X 26.3724,Y -65.4133,Z 79,A -72.8222,B 24.9043,C -2.2588,E1 25.0615,E2 517.1354} C_DIS
LIN {X 29.246,Y -64.1803,Z 79,A -70.0181,B 24.9034,C -2.2697,E1 25.0687,E2 514.3124} C_DIS
LIN {X 32.4844,Y -62.6043,Z 79,A -67.3016,B 24.9034,C -2.2688,E1 25.0755,E2 511.6054} C_DIS
LIN {X 34.7545,Y -61.3731,Z 79,A -65.3664,B 24.9034,C -2.268,E1 25.0802,E2 509.6777} C_DIS
LIN {X 36.9766,Y -60.0603,Z 79,A -63.1171,B 24.9028,C -2.2761,E1 25.0856,E2 507.4164} C_DIS
LIN {X 39.1812,Y -58.6461,Z 79,A -61.0035,B 24.9025,C -2.2798,E1 25.0905,E2 505.3009} C_DIS
LIN {X 41.4835,Y -57.0396,Z 79,A -58.7869,B 24.9022,C -2.2827,E1 25.0956,E2 503.0853} C_DIS
LIN {X 43.9933,Y -55.1276,Z 79,A -56.1921,B 24.9017,C -2.289,E1 25.1013,E2 500.485} C_DIS
LIN {X 46.393,Y -53.1229,Z 79,A -53.7604,B 24.9015,C -2.2917,E1 25.1065,E2 498.0564} C_DIS
LIN {X 48.6233,Y -51.0911,Z 79,A -51.2465,B 24.9008,C -2.2991,E1 25.1116,E2 495.5352} C_DIS
LIN {X 50.7639,Y -48.963,Z 79,A -48.9311,B 24.9006,C -2.3013,E1 25.1161,E2 493.2245} C_DIS
LIN {X 52.7658,Y -46.7998,Z 79,A -46.4429,B 24.8999,C -2.3099,E1 25.1208,E2 490.7271} C_DIS
LIN {X 54.7196,Y -44.4987,Z 79,A -44.078,B 24.8996,C -2.3138,E1 25.125,E2 488.3638} C_DIS
LIN {X 56.5069,Y -42.2062,Z 79,A -41.714,B 24.899,C -2.3202,E1 25.1291,E2 485.9961} C_DIS
LIN {X 58.1615,Y -39.8971,Z 79,A -39.4659,B 24.8986,C -2.3248,E1 25.1327,E2 483.748} C_DIS
LIN {X 59.5872,Y -37.7346,Z 79,A -37.2245,B 24.8977,C -2.3345,E1 25.1361,E2 481.4948} C_DIS
LIN {X 60.9325,Y -35.5213,Z 79,A -35.1305,B 24.8972,C -2.3402,E1 25.1391,E2 479.3981} C_DIS
LIN {X 62.2019,Y -33.2484,Z 79,A -33.1833,B 24.8972,C -2.3416,E1 25.1417,E2 477.4578} C_DIS
LIN {X 63.3777,Y -30.9483,Z 79,A -30.9501,B 24.8962,C -2.3516,E1 25.1445,E2 475.2129} C_DIS
LIN {X 64.4889,Y -28.5604,Z 79,A -28.7971,B 24.8956,C -2.3584,E1 25.1469,E2 473.0557} C_DIS
LIN {X 65.746,Y -25.532,Z 79,A -26.306,B 24.8954,C -2.3615,E1 25.1495,E2 470.5708} C_DIS
LIN {X 66.6929,Y -22.9476,Z 79,A -24.2311,B 24.8952,C -2.3638,E1 25.1515,E2 468.5021} C_DIS
LIN {X 67.4295,Y -20.6799,Z 79,A -22.1467,B 24.8942,C -2.374,E1 25.1532,E2 466.4055} C_DIS
LIN {X 68.2003,Y -17.9792,Z 79,A -19.766,B 24.8934,C -2.3839,E1 25.155,E2 464.015} C_DIS
LIN {X 68.8145,Y -15.4626,Z 79,A -17.6768,B 24.8928,C -2.3901,E1 25.1563,E2 461.9233} C_DIS
LIN {X 69.3408,Y -12.8991,Z 79,A -15.7174,B 24.8926,C -2.3921,E1 25.1573,E2 459.9707} C_DIS
LIN {X 69.7662,Y -10.3543,Z 79,A -13.4857,B 24.8917,C -2.4026,E1 25.1583,E2 457.7273} C_DIS
LIN {X 70.098,Y -7.7964,Z 79,A -11.4076,B 24.8911,C -2.4088,E1 25.159,E2 455.6469} C_DIS
LIN {X 70.3392,Y -5.1895,Z 79,A -9.2926,B 24.8905,C -2.4152,E1 25.1595,E2 453.5293} C_DIS
LIN {X 70.4819,Y -2.6132,Z 79,A -7.2044,B 24.8899,C -2.4217,E1 25.1597,E2 451.4382} C_DIS
LIN {X 70.5283,Y 0.3427,Z 79,A -4.9578,B 24.8896,C -2.4249,E1 25.1597,E2 449.1974} C_DIS
LIN {X 70.4554,Y 3.2295,Z 79,A -2.7416,B 24.8893,C -2.4286,E1 25.1596,E2 446.9855} C_DIS
LIN {X 70.3239,Y 5.3815,Z 79,A -0.8198,B 24.8884,C -2.439,E1 25.1592,E2 445.0507} C_DIS
LIN {X 70.0401,Y 8.2909,Z 79,A 1.397,B 24.8881,C -2.442,E1 25.1585,E2 442.84} C_DIS
LIN {X 69.7344,Y 10.5601,Z 79,A 3.3791,B 24.8872,C -2.4512,E1 25.1577,E2 440.8476} C_DIS
LIN {X 69.2207,Y 13.5233,Z 79,A 5.6311,B 24.887,C -2.4533,E1 25.1566,E2 438.6038} C_DIS
LIN {X 68.6804,Y 16.0433,Z 79,A 7.8548,B 24.8861,C -2.4634,E1 25.1552,E2 436.3692} C_DIS
LIN {X 67.9756,Y 18.811,Z 79,A 10.2598,B 24.8852,C -2.4728,E1 25.1535,E2 433.9559} C_DIS
LIN {X 67.24,Y 21.2911,Z 79,A 12.1438,B 24.8852,C -2.4728,E1 25.152,E2 432.0824} C_DIS
LIN {X 66.4142,Y 23.7417,Z 79,A 14.4263,B 24.8842,C -2.4842,E1 25.1499,E2 429.7861} C_DIS
LIN {X 65.4046,Y 26.3938,Z 79,A 16.6546,B 24.8838,C -2.4886,E1 25.1476,E2 427.5596} C_DIS
LIN {X 64.2144,Y 29.1702,Z 79,A 18.9333,B 24.8836,C -2.4907,E1 25.145,E2 425.2885} C_DIS
LIN {X 63.2807,Y 31.1439,Z 79,A 20.8515,B 24.8827,C -2.4996,E1 25.1427,E2 423.3594} C_DIS
LIN {X 61.9057,Y 33.7945,Z 79,A 23.0959,B 24.8826,C -2.5011,E1 25.1398,E2 421.1232} C_DIS
LIN {X 60.8389,Y 35.6796,Z 79,A 25.0239,B 24.8817,C -2.5105,E1 25.1371,E2 419.1832} C_DIS
LIN {X 59.2706,Y 38.2278,Z 79,A 27.2764,B 24.8816,C -2.5118,E1 25.1337,E2 416.9389} C_DIS
LIN {X 57.7901,Y 40.4314,Z 79,A 29.5332,B 24.8808,C -2.52,E1 25.1302,E2 414.6739} C_DIS
LIN {X 56.1349,Y 42.7013,Z 79,A 31.8609,B 24.8802,C -2.5267,E1 25.1263,E2 412.3414} C_DIS
LIN {X 54.3133,Y 44.9936,Z 79,A 34.1627,B 24.8798,C -2.5302,E1 25.1222,E2 410.0421} C_DIS
LIN {X 52.3381,Y 47.2776,Z 79,A 36.7148,B 24.879,C -2.5384,E1 25.1175,E2 407.4819} C_DIS
LIN {X 50.1891,Y 49.552,Z 79,A 39.1609,B 24.8788,C -2.5413,E1 25.1128,E2 405.0397} C_DIS
LIN {X 48.0048,Y 51.6728,Z 79,A 41.7486,B 24.878,C -2.5494,E1 25.1075,E2 402.4434} C_DIS
LIN {X 45.7341,Y 53.6912,Z 79,A 44.1792,B 24.8776,C -2.5532,E1 25.1024,E2 400.0134} C_DIS
LIN {X 43.3941,Y 55.6011,Z 79,A 46.6201,B 24.8772,C -2.5572,E1 25.097,E2 397.5719} C_DIS
LIN {X 41.325,Y 57.1557,Z 79,A 48.7014,B 24.8769,C -2.5603,E1 25.0924,E2 395.4908} C_DIS
LIN {X 39.0011,Y 58.7649,Z 79,A 50.9318,B 24.8768,C -2.5623,E1 25.0872,E2 393.2633} C_DIS
LIN {X 36.4504,Y 60.3801,Z 79,A 53.2,B 24.8768,C -2.5611,E1 25.0818,E2 391.0052} C_DIS
LIN {X 34.2079,Y 61.6783,Z 79,A 55.2993,B 24.8766,C -2.5638,E1 25.0768,E2 388.9055} C_DIS
LIN {X 32.3379,Y 62.6792,Z 79,A 57.2235,B 24.8759,C -2.5714,E1 25.072,E2 386.9689} C_DIS
LIN {X 29.5786,Y 64.0273,Z 79,A 59.505,B 24.8761,C -2.5688,E1 25.0662,E2 384.6995} C_DIS
LIN {X 27.6107,Y 64.9003,Z 79,A 61.4332,B 24.8755,C -2.5753,E1 25.0613,E2 382.7604} C_DIS
LIN {X 24.8277,Y 66.0149,Z 79,A 63.6856,B 24.8757,C -2.5729,E1 25.0554,E2 380.5186} C_DIS
LIN {X 22.4583,Y 66.8579,Z 79,A 65.9164,B 24.8751,C -2.5795,E1 25.0495,E2 378.2766} C_DIS
LIN {X 19.6357,Y 67.7419,Z 79,A 68.3634,B 24.8748,C -2.5824,E1 25.043,E2 375.8272} C_DIS
LIN {X 16.9553,Y 68.4611,Z 79,A 70.5625,B 24.8748,C -2.5824,E1 25.037,E2 373.6315} C_DIS
LIN {X 13.983,Y 69.1294,Z 79,A 72.8423,B 24.8752,C -2.5785,E1 25.0308,E2 371.3636} C_DIS
LIN {X 11.8592,Y 69.5253,Z 79,A 74.778,B 24.8747,C -2.5837,E1 25.0255,E2 369.4176} C_DIS
LIN {X 8.8791,Y 69.9682,Z 79,A 77.0499,B 24.875,C -2.5799,E1 25.0192,E2 367.1568} C_DIS
LIN {X 6.2748,Y 70.2497,Z 79,A 79.1693,B 24.875,C -2.5799,E1 25.0134,E2 365.0386} C_DIS
LIN {X 3.6956,Y 70.4325,Z 79,A 81.2714,B 24.875,C -2.58,E1 25.0075,E2 362.9373} C_DIS
LIN {X 1.1135,Y 70.5205,Z 79,A 83.4906,B 24.8748,C -2.5828,E1 25.0013,E2 360.712} C_DIS
LIN {X -1.7299,Y 70.5092,Z 79,A 85.9293,B 24.8745,C -2.5854,E1 24.9945,E2 358.267} C_DIS
LIN {X -4.3155,Y 70.3982,Z 79,A 87.8782,B 24.8749,C -2.5809,E1 24.9891,E2 356.3283} C_DIS
LIN {X -6.8945,Y 70.1925,Z 79,A 90.0667,B 24.8749,C -2.582,E1 24.983,E2 354.1361} C_DIS
LIN {X -9.4839,Y 69.8898,Z 79,A 92.1035,B 24.8752,C -2.5788,E1 24.9773,E2 352.1055} C_DIS
LIN {X -12.0615,Y 69.4914,Z 79,A 94.3796,B 24.8749,C -2.5811,E1 24.971,E2 349.8217} C_DIS
LIN {X -14.6023,Y 69.0022,Z 79,A 96.4859,B 24.8751,C -2.5794,E1 24.9653,E2 347.7169} C_DIS
LIN {X -17.3336,Y 68.3663,Z 79,A 98.7034,B 24.8754,C -2.5758,E1 24.9593,E2 345.5049} C_DIS
LIN {X -20.2363,Y 67.5639,Z 79,A 101.2103,B 24.8755,C -2.5747,E1 24.9526,E2 342.9966} C_DIS
LIN {X -23.1471,Y 66.6229,Z 79,A 103.6443,B 24.876,C -2.5705,E1 24.9461,E2 340.5681} C_DIS
LIN {X -25.9775,Y 65.5711,Z 79,A 105.9376,B 24.8766,C -2.5635,E1 24.9402,E2 338.2866} C_DIS
LIN {X -27.9965,Y 64.7348,Z 79,A 107.8816,B 24.8765,C -2.565,E1 24.9352,E2 336.3346} C_DIS
LIN {X -30.7338,Y 63.4809,Z 79,A 110.1605,B 24.8772,C -2.5573,E1 24.9294,E2 334.0681} C_DIS
LIN {X -33.0381,Y 62.3127,Z 79,A 112.269,B 24.8775,C -2.5542,E1 24.9242,E2 331.9615} C_DIS
LIN {X -35.2958,Y 61.0622,Z 79,A 114.4917,B 24.8775,C -2.5534,E1 24.9188,E2 329.734} C_DIS
LIN {X -37.685,Y 59.6182,Z 79,A 116.91,B 24.8777,C -2.5527,E1 24.913,E2 327.3098} C_DIS
LIN {X -39.9168,Y 58.1478,Z 79,A 119.0732,B 24.8781,C -2.5483,E1 24.908,E2 325.1499} C_DIS
LIN {X -42.0197,Y 56.6469,Z 79,A 121.1577,B 24.8785,C -2.5438,E1 24.9033,E2 323.069} C_DIS
LIN {X -44.4022,Y 54.7977,Z 79,A 123.6512,B 24.8789,C -2.5396,E1 24.8979,E2 320.5762} C_DIS
LIN {X -46.7838,Y 52.7802,Z 79,A 126.1772,B 24.8795,C -2.5337,E1 24.8926,E2 318.0543} C_DIS
LIN {X -48.942,Y 50.7842,Z 79,A 128.6079,B 24.8799,C -2.5291,E1 24.8876,E2 315.6246} C_DIS
LIN {X -51.0788,Y 48.6363,Z 79,A 131.0994,B 24.8804,C -2.5238,E1 24.8828,E2 313.135} C_DIS
LIN {X -53.1081,Y 46.41,Z 79,A 133.5334,B 24.881,C -2.5175,E1 24.8783,E2 310.7052} C_DIS
Enddeposition()
END
